// TIA Portal project "CGS1218_000_40" (V16)

(* hardware
DEVICE "SIMATIC 300"  S7-300 station
   slot 0: "Rack 0"  Rail  6ES7 390-1***0-0AA0
   slot 2: "CPU 317-2 PN/DP"  Unspecific CPU S7 300  6ES7 3XX-XXXXX-XXXX
DEVICE "SLIO_SLAVE"  S7-300 station
   slot 0: "Rack 0"  Rail  6ES7 390-1***0-0AA0
   slot 2: "CPU 315-2 PN/DP"  Unspecific CPU S7 300  6ES7 3XX-XXXXX-XXXX
DEVICE "Rack 0"  S7-300 station
   slot 0: "Rail_0"  Rail  6ES7 390-1***0-0AA0
   slot 2: "Mig_PVA_AWL"  Unspecific CPU S7 300  6ES7 3XX-XXXXX-XXXX
*)

// ===== PLC "CPU 317-2 PN/DP"  Unspecific CPU S7 300 =====
// protected blocks, not shown: "AG_LRECV_LF", "AG_LSEND_LF", "AG_RECV", "AG_SEND", "DCO_ReadDriveParameter", "DCO_WriteDriveParameter", "GLOBAL_DP_DIAG", "IO_LINK_DEVICE", "IO_LINK_MASTER"

VAR_GLOBAL   // PLC tag table "STEP7 classic symbols"
   "HDI_LS_FCH_LFT_DN" AT %I32.1 : Bool;   // HDI def M 88.1: limit switch furnace chamber lift down
   "HDI_LS_GCH_BEL_DN" AT %I274.7 : Bool;   // HDI def M 97.7: limit switch gate chamber bellow in lower position
   "HDO_XT_CLP_BLW_BRK" AT %Q275.2 : Bool;   // HDO def M 164.2: Brake crystal clamp below
   "HDO_XT_CLP_BLW_CL" AT %Q275.1 : Bool;   // HDO def M 164.1: Motor crystal clamp below close
   "HDO_XT_CLP_BLW_OP" AT %Q275.0 : Bool;   // HDO def M 164.0: Motor crystal clamp below open
   "HDO_XT_CLP_BLW_RST" AT %Q275.3 : Bool;   // HDO def M 164.3: Reset controller crystal clamp below
   "HDO_XT_CLP_TILT_BRK" AT %Q274.2 : Bool;   // HDO def M 163.2: Motor crystal clamp tilt brake
   "HDO_XT_CLP_TILT_BW" AT %Q274.0 : Bool;   // HDO def M 163.0: Motor crystal clamp tilt backwards
   "HDO_XT_CLP_TILT_FW" AT %Q274.1 : Bool;   // HDO def M 163.1: Motor crystal clamp tilt forwards (75?
   "HDO_XT_DRP_OUT_PRT_CL" AT %Q224.6 : Bool;   // HDO def M 150.6: Valve block close crystal drop out protection
   "HDO_XT_DRP_OUT_PRT_OP" AT %Q224.7 : Bool;   // HDO def M 150.7: Valve block open crystal drop out protection
   "HDO_XT_HDL_LFT_ENB" AT %Q272.7 : Bool;   // HDO def M 160.7: controller enable crystal handling lift
   "HDO_XT_HDL_SLID_BW" AT %Q273.7 : Bool;   // HDO def M 161.7: Motor crystal handling slider backwards
   "HDO_XT_HDL_SLID_FW" AT %Q273.6 : Bool;   // HDO def M 161.6: Motor crystal handling slider forwards
   "HDO_XT_HDL_SW_ENB" AT %Q273.0 : Bool;   // HDO def M 161.0: controller enable crystal handling swivel
   "HDO_XT_HDL_SW_LOCK" AT %Q225.4 : Bool;   // HDO def M 151.4: Valve block xtal handling swivel lock close (145?
   "HDO_XT_HDL_SW_UNLOCK" AT %Q225.5 : Bool;   // HDO def M 151.5: Valve block xtal handling swivel lock open (145?
   "HDO_XT_LFT_ENB" AT %Q272.6 : Bool;   // HDO def M 160.6: controller enable crystal lift
   "SM_TMR_PWR_FAIL_5S" AT %T150 : Timer;   // main line power fail 5 sec
   "STA_ITL_CAUSE" AT %MW20 : Word;
   "STA_ITL_CAUSE_DLY" AT %MW22 : Int;
   "STA_ITL_NO" AT %MB20 : Byte;
   "STA_ITL_STAT" AT %MB21 : Byte;
   "P_STA_WTR_VAC_BYP" AT %IW2194 : Word;
   "P_STA_WTR_BCH" AT %IW2164 : Word;
   "P_STA_WTR_CFT_B" AT %IW2188 : Word;
   "P_STA_WTR_CR_SFT" AT %IW2020 : Word;
   "P_STA_WTR_CUR_FEED" AT %IW2182 : Word;
   "P_STA_WTR_FCH" AT %IW2146 : Word;
   "P_STA_WTR_GCH" AT %IW2050 : Word;
   "P_STA_WTR_GCH_ADDS" AT %IW2086 : Word;
   "P_STA_WTR_GCH_H" AT %IW2068 : Word;
   "P_STA_WTR_GCH_V" AT %IW2074 : Word;
   "P_BM_MAG_ACT_CUR" AT %IW868 : Word;
   "P_BM_MAG_ACT_TMP_COIL_A1" AT %IW872 : Word;
   "P_BM_MAG_ACT_TMP_COIL_A2" AT %IW874 : Word;
   "P_BM_MAG_ACT_TMP_COIL_B1" AT %IW876 : Word;
   "P_BM_MAG_ACT_TMP_COIL_B2" AT %IW878 : Word;
   "P_BM_MAG_ACT_TMP_SHLD" AT %IW880 : Word;
   "P_BM_MAG_ACT_VLT" AT %IW870 : Word;
   "P_BM_MAG_CTRL" AT %QB864 : Byte;
   "P_BM_MAG_SET_CUR" AT %QW865 : Word;
   "P_BM_MAG_STAT" AT %IB864 : Byte;
   "P_BM_MAG_STAT2" AT %IW865 : Word;
   "P_BM_MAG_STAT3" AT %IB867 : Byte;
   "BM_MCC_OFF_TME" AT %T132 : Timer;   // melt contact control off time
   "HDI_ACC_UPS_24V_NRM" AT %I89.7 : Bool;   // HDI def M 93.7: ACC UPS Alarm
   "HDI_ACC_WTR_FLW_IN_OK" AT %I88.4 : Bool;   // HDI def M 92.4: ACC input waterflow ok
   "HDI_ACC_WTR_FLW_OUT_OK" AT %I88.3 : Bool;   // HDI def M 92.3: ACC output waterflow ok
   "HDI_ACC_WTR_TMP_OUT_OK" AT %I88.5 : Bool;   // HDI def M 92.5: ACC output watertemp. Ok
   "HDI_CB_FLT_AC230V" AT %I16.3 : Bool;   // HDI def M 72.3: fault circuit breakers AC 230V 1=OK
   "HDI_CB_FLT_AC400V_K2" AT %I16.1 : Bool;   // HDI def M 72.1: fault circuit breakers AC 400V 1=OK
   "HDI_CB_FLT_AC400V_K5" AT %I34.0 : Bool;   // HDI def M 90.0: fault circuit breakers AC 400V +K5 1=OK
   "HDI_CB_FLT_AC400V_K8" AT %I277.6 : Bool;   // HDI def M 100.6: fault circuit breakers AC 400V 1=OK
   "HDI_CB_FLT_DC24V_K2" AT %I16.0 : Bool;   // HDI def M 72.0: fault circuit breakers DC 24V 1=OK
   "HDI_CB_FLT_DC24V_K5" AT %I34.1 : Bool;   // HDI def M 90.1: fault circuit breakers DC 24V +K5 1=OK
   "HDI_CB_FLT_DC24V_K8" AT %I277.7 : Bool;   // HDI def M 100.7: fault circuit breakers DC 24V 1=OK
   "HDI_COMP_AIR_2_OK" AT %I35.7 : Bool;   // HDI def M 91.7: pressure switch compressed air 2 (ACC) ok
   "HDI_COMP_AIR_OK" AT %I35.6 : Bool;   // HDI def M 91.6: pressure switch compressed air ok
   "HDI_DPH_RPT_DET_OK" AT %I90.0 : Bool;   // HDI def M 94.0: ACC Diaphraghm rupture detector OK
   "HDI_EMO" AT %I17.3 : Bool;   // HDI def M 73.3: Emergency off (1=ok)
   "HDI_EMS" AT %I17.4 : Bool;   // HDI def M 73.4: Emergency stop handling drives (1=ok)
   "HDI_MP_ENB_K5" AT %I35.3 : Bool;   // HDI def M 91.3: Mobile panel agree button +K5
   "HDI_MP_ENB_K8" AT %I279.6 : Bool;   // HDI def M 102.6: Mobile panel agree button +K8
   "HDI_MP_ENB_K9" AT %I279.7 : Bool;   // HDI def M 102.7: Mobile panel agree button +K9
   "HDI_OIL_LVL_CR_SFT" AT %I35.0 : Bool;   // HDI def M 91.0: Crucible shaft min. oil level
   "HDI_OIL_LVL_XT_SFT" AT %I279.1 : Bool;   // HDI def M 102.1: Crystal shaft min. oil level
   "HDI_OV_PRS_1_FLT" AT %I88.6 : Bool;   // HDI def M 92.6: ACC overpressure 1 error/fault
   "HDI_OV_PRS_2_FLT" AT %I88.7 : Bool;   // HDI def M 92.7: ACC overpressure 2 error/fault
   "HDI_P1_FLT" AT %I18.1 : Bool;   // HDI def M 74.1: pump unit (P1) error
   "HDI_P1_IS_ON" AT %I18.2 : Bool;   // HDI def M 74.2: pump unit (P1) running
   "P_BM_UP_FCH_SW_ENC_REF" AT %QD1184 : DWord;   // Setpoint reference position upper furnace chamber swivel
   "BM_VAC_TMR_APS_BY_FIL" AT %T102 : Timer;   // Timer for delayed APS bypass filter
   "BM_VAC_TMR_APS_FCH" AT %T101 : Timer;   // Timer for delayed APS furnace
   "BM_VAC_TMR_APS_FDR" AT %T99 : Timer;   // Timer for delayed APS feeder
   "BM_VAC_TMR_APS_FIL" AT %T98 : Timer;   // Timer for delayed APS main filter
   "BM_VAC_TMR_APS_GCH" AT %T100 : Timer;   // Timer for delayed APS gate
   "BM_VAC_TMR_V2_ON" AT %T104 : Timer;   // Timer for delayed opening V2 after P1 on
   "BM_VAC_TMR_V3_ON" AT %T105 : Timer;   // Timer for delayed opening V3 after P3 on
   "HDI_LS_V3_OP" AT %I280.0 : Bool;   // HDI def M 103.0: valve position V3 open
   "HDI_LS_V7_CLN_POS" AT %I274.5 : Bool;   // HDI def M 97.5: limit switch gate valve V7 in cleaning position
   "HDI_LS_V7_DN" AT %I274.1 : Bool;   // HDI def M 97.1: limit switch gate valve V7 in lower position
   "HDI_LS_V7_FLP_OP" AT %I274.4 : Bool;   // HDI def M 97.4: limit switch gate valve V7 flap open
   "HDI_LS_V7_SW_IN" AT %I274.2 : Bool;   // HDI def M 97.2: limit switch gate valve V7 swiveled in
   "HDI_LS_V7_SW_OUT" AT %I274.3 : Bool;   // HDI def M 97.3: limit switch gate valve V7 swiveled out
   "HDO_SPARE_18_4" AT %Q18.4 : Bool;   // HDO def M 138.4: spare digital output
   "HDO_SPARE_18_5" AT %Q18.5 : Bool;   // HDO def M 138.5: spare digital output
   "HDO_SPARE_18_6" AT %Q18.6 : Bool;   // HDO def M 138.6: spare digital output
   "HDO_SPARE_18_7" AT %Q18.7 : Bool;   // HDO def M 138.7: spare digital output
   "HDO_SPARE_226_2" AT %Q226.2 : Bool;   // HDO def M 152.2: Valve block spare output
   "HDO_SPARE_226_3" AT %Q226.3 : Bool;   // HDO def M 152.3: Valve block spare output
   "HDO_SPARE_226_4" AT %Q226.4 : Bool;   // HDO def M 152.4: Valve block spare output
   "HDO_SPARE_226_5" AT %Q226.5 : Bool;   // HDO def M 152.5: Valve block spare output
   "HDO_SPARE_226_6" AT %Q226.6 : Bool;   // HDO def M 152.6: Valve block spare output
   "HDO_SPARE_226_7" AT %Q226.7 : Bool;   // HDO def M 152.7: Valve block spare output
   "P_BM_ACT_WTR_TMP_PWR_CAB" AT %IW2024 : Word;   // HAI def MW 356: actual water temperature high current cables Main K18
   "P_BM_ACT_WTR_TMP_PWR_CAB2" AT %IW2030 : Word;   // HAI def MW 347: actual water temperature current feed throughs B K19
   "P_BM_ACT_WTR_TMP_SOC_BCH" AT %IW2174 : Word;   // HAI def MW 329: actual water temperature socket bottom chamber K13
   "P_BM_ACT_WTR_TMP_TCH" AT %IW2090 : Word;   // HAI def MW 239: actual water temperature top chamber K07
   "P_BM_ACT_WTR_TMP_TEC_FLG" AT %IW2114 : Word;   // HAI def MW 275: actual water temperature technolity chamber K08
   "P_BM_ACT_WTR_TMP_UP_FCH" AT %IW2132 : Word;   // HAI def MW 338: actual water temperature upper furnace chamber K10
   "P_BM_ACT_WTR_TMP_VPTS" AT %IW2078 : Word;   // HAI def MW 291: actual water temperature view ports K06
   "P_BM_ACT_WTR_TMP_XT_SFT" AT %IW2036 : Word;   // HAI def MW 246: actual water temperature seed shaft K02
   "DP_DEATV_ERR_CODE_N9" AT %MW62 : Int;   // DP Slave +N9 (active cooling) deactivation error code
   "DP_DEATV_TSK_RUN_N9" AT %M52.5 : Bool;   // DP Slave +N9 (active cooling) deactivation busy flag
   "HDO_MAG_LFT_UP" AT %Q33.2 : Bool;   // HDO def M 143.2: Magnet lift drive upwards
   "HDO_MCC_ENB_XT" AT %Q275.5 : Bool;   // HDO def M 164.5: seed contact detection enable output (xt isolated)
   "HDO_MCC_TEST_XT" AT %Q275.4 : Bool;   // HDO def M 164.4: seed contact detection test output ( xt isolated)
   "HDO_MON_TMP_P2_RES" AT %Q17.7 : Bool;   // HDO def M 137.7: temperature monitoring pump 2 reset
   "HDO_P1_ON" AT %Q17.0 : Bool;   // HDO def M 137.0: Vacuum pump 1 on (furnace chamber)
   "HDO_P1_SEAL_GAS" AT %Q17.3 : Bool;   // HDO def M 137.3: Vacuum pump 1 seal gas on
   "HDO_P2_FU_ON" AT %Q144.0 : Bool;   // HDO def M 152.0: Frequency converter P2 start
   "HDO_P2_FU_RES" AT %Q144.1 : Bool;   // HDO def M 152.1: Frequency converter P2 fault reset
   "HDI_SPARE_16_5" AT %I16.5 : Bool;   // HDI def M 72.5: spare digital input
   "HDI_SPARE_16_6" AT %I16.6 : Bool;   // HDI def M 72.6: spare digital input
   "HDI_SPARE_16_7" AT %I16.7 : Bool;   // HDI def M 72.7: spare digital input
   "HDI_SPARE_17_0" AT %I17.0 : Bool;   // HDI def M 73.0: spare digital input
   "HDI_SPARE_17_5" AT %I17.5 : Bool;   // HDI def M 73.5: spare digital input
   "HDI_SPARE_17_6" AT %I17.6 : Bool;   // HDI def M 73.6: spare digital input
   "HDI_SPARE_17_7" AT %I17.7 : Bool;   // HDI def M 73.7: spare digital input
   "HDI_SPARE_18_7" AT %I18.7 : Bool;   // HDI def M 74.7: spare digital input
   "HDI_SPARE_275_7" AT %I275.7 : Bool;   // HDI def M 98.7: spare digital input
   "HDI_SPARE_280_5" AT %I280.5 : Bool;   // HDI def M 103.5: spare digital input
   "HDI_SPARE_280_6" AT %I280.6 : Bool;   // HDI def M 103.6: spare digital input
   "HDI_SPARE_280_7" AT %I280.7 : Bool;   // HDI def M 103.7: spare digital input
   "HDI_SPARE_33_4" AT %I33.4 : Bool;   // HDI def M 89.4: spare
   "HDI_SPARE_33_5" AT %I33.5 : Bool;   // HDI def M 89.5: spare
   "HDI_SPARE_48_2" AT %I88.2 : Bool;   // HDI def M 92.2: ACC spare
   "HDI_SPARE_90_2" AT %I90.2 : Bool;   // HDI def M 94.2: ACC spare
   "P_reserve_2_X08_WTR_TMP" AT %IW2108 : Word;
   "P_reserve_3_X08_WTR_FLW" AT %IW2154 : Word;
   "HDI_LS_V2_11_OP" AT %I36.6 : Bool;   // HDI def M 105.6: limit switch valve v2.11 opened
   "HDI_LS_V2_1_CL" AT %I33.7 : Bool;   // HDI def M 89.7: valve position v2.1 fce chamber
   "HDI_LS_V2_1_OP" AT %I33.6 : Bool;   // HDI def M 89.6: valve position v2.1 fce chamber
   "HDI_LS_V3_3_CL" AT %I36.5 : Bool;   // HDI def M 105.5: limit switch valve v3.3 closed
   "HDI_LS_V3_3_OP" AT %I36.4 : Bool;   // HDI def M 105.4: limit switch valve v3.3 opened
   "HDI_LS_V3_4_CL" AT %I36.3 : Bool;   // HDI def M 105.3: limit switch valve v3.4 closed
   "HDI_LS_V3_4_OP" AT %I36.2 : Bool;   // HDI def M 105.2: limit switch valve v3.4 opened
   "HDI_LS_V3_CL" AT %I280.1 : Bool;   // HDI def M 103.1: Valve position V3 closed
   "MELT_CON_DETECT_DLY" AT %T134 : Timer;   // melt contact control delay timer
   "SysEdgeFlag400ms" AT %M3.4 : Bool;   // System Cycle: Edge Flag 400 ms
   "SysEdgeFlag500ms" AT %M3.6 : Bool;   // System Cycle: Edge Flag 500 ms
   "SysEdgeFlag800ms" AT %M4.0 : Bool;   // System Cycle: Edge Flag 800 ms
   "SysImpFlag100ms" AT %M3.1 : Bool;   // System Cycle: Impuls Flag 100 ms
   "SysImpFlag1_6s" AT %M4.5 : Bool;   // System Cycle: Impuls Flag 1600 ms
   "SysImpFlag1s" AT %M4.3 : Bool;   // System Cycle: Impuls Flag 1000 ms
   "SysImpFlag200ms" AT %M3.3 : Bool;   // System Cycle: Impuls Flag 200 ms
   "SysImpFlag2s" AT %M4.7 : Bool;   // System Cycle: Impuls Flag 2000 ms
   "SysImpFlag400ms" AT %M3.5 : Bool;   // System Cycle: Impuls Flag 400 ms
   "SysImpFlag500ms" AT %M3.7 : Bool;   // System Cycle: Impuls Flag 500 ms
   "SysImpFlag800ms" AT %M4.1 : Bool;   // System Cycle: Impuls Flag 800 ms
   "SysLog0" AT %M0.0 : Bool;   // System: Logical 0
   "SysLog1" AT %M0.1 : Bool;   // System: Logical 1
   "SysTick100ms" AT %M1.0 : Bool;   // System Tick: 100 ms
   "P_BM_PWR_SPL_2_SET_PWR" AT %QD902 : Real;   // setpoint power heater 2
   "P_BM_PWR_SPL_CTRL" AT %QB896 : Byte;   // Heater on
   "P_BM_PWR_SPL_CTRL_W" AT %QW896 : Word;   // power supply control word
   "P_BM_PWR_SPL_STAT" AT %IW896 : Word;   // statusword 1 power supply
   "P_BM_PWR_SPL_STAT2" AT %IW898 : Word;   // statusword 2 power supply
   "P_BM_PWR_SPL_STAT3" AT %IW900 : Word;   // statusword 3 power supply
   "P_BM_PWR_SPL_STAT4" AT %IW902 : Word;   // statusword 4 power supply
   "P_BM_PWR_SPL_STAT5" AT %IW904 : Word;   // statusword 5 power supply
   "P_BM_PWR_SPL_STAT6" AT %IW906 : Word;   // statusword 6 power supply
   "P_BM_PWR_SPL_STAT7" AT %IW908 : Word;   // statusword 7 power supply
   "HDI_LS_MAG_LFT_UP" AT %I34.2 : Bool;   // HDI def M 90.2: limit switch magnet lift up
   "HDI_LS_TCH_DN" AT %I273.0 : Bool;   // HDI def M 96.0: limit switch top chamber in lower position
   "HDI_LS_TCH_SW_CLN" AT %I273.2 : Bool;   // HDI def M 96.2: limit switch top chamber swivelled in cleaning pos
   "HDI_LS_TCH_SW_IN" AT %I273.1 : Bool;   // HDI def M 96.1: limit switch top chamber swivelled in
   "HDI_LS_TCH_SW_LOCK" AT %I273.4 : Bool;   // HDI def M 96.4: limit switch top chamber swivel locked
   "HDI_LS_TCH_SW_OUT" AT %I273.3 : Bool;   // HDI def M 96.3: limit switch top chamber swivelled out
   "HDI_LS_TCH_TILT_0" AT %I273.5 : Bool;   // HDI def M 96.5: limit switch top chamber tilt 0?horizental
   "HDI_LS_TCH_TILT_30" AT %I273.6 : Bool;   // HDI def M 96.6: limit switch top chamber tilt 30?Cleaning position
   "HDI_LS_TCH_UP" AT %I272.7 : Bool;   // HDI def M 95.7: limit switch top chamber in upper position
   "HDI_LS_TEC_FLG_DN" AT %I32.4 : Bool;   // HDI def M 88.4: limit switch technolgy flange down
   "HDO_HOR_OPP_K2" AT %Q16.0 : Bool;   // HDO def M 136.0: Horn +K2
   "HDO_HOR_OPP_K8" AT %Q272.0 : Bool;   // HDO def M 160.0: Horn +K8
   "HDO_HOR_OPP_K9" AT %Q276.3 : Bool;   // HDO def M 165.3: Horn +K9
   "HDO_HTR_PWR_ON" AT %Q17.5 : Bool;   // HDO def M 137.4: Heater power supply on
   "P_BM_ACT_GAS_FLW_MFC_1" AT %ID1376 : Real;   // actual gas flow from mfc with profinet interface
   "P_BM_ACT_GAS_FLW_MFC_2" AT %ID1408 : Real;   // actual gas flow from mfc with profinet interface
   "P_BM_ACT_WTR_FLW_VAC_BYP" AT %IW2190 : Word;   // actual water flow vacuum bypass tube
   "P_BM_ACT_WTR_FLW_BCH" AT %IW2160 : Word;   // HAI def MW 309: actual water flow bottom chamber K12
   "P_BM_ACT_WTR_FLW_CFT_B" AT %IW2184 : Word;   // HAI def MW 235: actual water flow current feed throught Bot K15
   "P_BM_ACT_WTR_FLW_CFT_M" AT %IW2178 : Word;   // HAI def MW 217: actual water flow current feed throught Main K14
   "P_BM_ACT_WTR_FLW_CR_SFT" AT %IW2016 : Word;   // HAI def MW 208: actual water flow crucible shaft K17
   "P_BM_ACT_WTR_FLW_FCH" AT %IW2142 : Word;   // HAI def MW 300: actual water flow furnace chamber K11
   "P_BM_ACT_WTR_FLW_GCH" AT %IW2046 : Word;   // HAI def MW 262: actual water flow gate chamber K03
   "P_BM_ACT_WTR_FLW_GCH_ADDS" AT %IW2082 : Word;   // HAI def MW 298: actual water flow chamber parts, view ports K24
   "HDI_XT_ROT_CAM_TRG" AT %I279.5 : Bool;   // HDI def M 102.5: limit switch xtal rotation camera trigger
   "HDO_ACC_ALM_LT_1" AT %Q88.4 : Bool;   // HDO def M 146.4: ACC Blitzlicht Kasten
   "HDO_ACC_ALM_LT_2" AT %Q88.6 : Bool;   // HDO def M 146.6: ACC Blitzlicht Bedienpult
   "HDO_ACC_ALM_SND_1" AT %Q88.5 : Bool;   // HDO def M 146.5: ACC Sirene Kasten
   "HDO_ACC_ALM_SND_2" AT %Q88.7 : Bool;   // HDO def M 146.7: ACC Sirene Bedienpult
   "HDO_ACC_SC_HTR_RST" AT %Q88.1 : Bool;   // HDO def M 146.1: ACC Heizung RESET
   "HDO_ACC_SC_HTR_STR" AT %Q88.0 : Bool;   // HDO def M 146.0: ACC Heizung START
   "HDO_ACC_SC_WTR_RST" AT %Q88.3 : Bool;   // HDO def M 146.3: ACC K黨lwasser RESET
   "HDO_ACC_SC_WTR_STR" AT %Q88.2 : Bool;   // HDO def M 146.2: ACC K黨lwasser START
   "HDO_BEL_LFT_ENB" AT %Q276.2 : Bool;   // HDO def M 165.2: controller enable gate bellow lift
   "HDO_BRK_MAG_LFT" AT %Q33.4 : Bool;   // HDO def M 143.4: Brake magnet lift
   "HDO_CR_LFT_ENB" AT %Q32.6 : Bool;   // HDO def M 142.6: controller enable crucible lift
   "HDO_CR_ROT_ENB" AT %Q32.5 : Bool;   // HDO def M 142.5: controller enable crucible rotation
   "HDO_FCH_HOOK_HOME" AT %Q96.0 : Bool;   // HDO def M 150.0: Valve block lower furnace chamber hook unlocking
   "HDO_V24" AT %Q224.5 : Bool;   // HDO def M 150.5: Valve block V24 valve argon gas inlet feeder
   "HDO_V25" AT %Q96.5 : Bool;   // HDO def M 150.5: Valve block argon inlet pressure storage tank, V25 open
   "HDO_V2_1" AT %Q96.6 : Bool;   // HDO def M 150.6: Valve block vacuum valve, V2.1 open
   "HDO_V2_11" AT %Q97.7 : Bool;   // HDO def M 151.7: Valve block vacuum valve, V2.11 open
   "HDO_V3" AT %Q224.3 : Bool;   // HDO def M 150.3: Valve block V3 vacuum valve (gate chamber)
   "HDO_V3_2" AT %Q224.4 : Bool;   // HDO def M 150.4: Valve block V3.2 vacuum valve feeder
   "HDO_V3_3" AT %Q97.6 : Bool;   // HDO def M 151.6: Valve block vacuum valve, V3.3 open
   "HDO_V3_4" AT %Q97.5 : Bool;   // HDO def M 151.5: Valve block vacuum valve, V3.4 open
   "HDO_V4" AT %Q224.0 : Bool;   // HDO def M 150.0: Valve block V4 valve argon gas inlet (gate chamber)
   "HDO_V5" AT %Q224.1 : Bool;   // HDO def M 150.1: Valve block V5 valve argon gas inlet controlled (gch)
   "HDO_V6" AT %Q224.2 : Bool;   // HDO def M 150.2: Valve block V6 valve argon gas inlet controlled (Fch)
   "HDO_V9_2" AT %Q97.3 : Bool;   // HDO def M 151.3: Valve block ventiliation valve vaccum line gate, V9_2
   "HDO_XT_CLP_ABV_BRK" AT %Q274.5 : Bool;   // HDO def M 163.5: Brake crystal clamp above
   "HDO_XT_CLP_ABV_CL" AT %Q274.4 : Bool;   // HDO def M 163.4: Motor crystal clamp above close
   "HDO_XT_CLP_ABV_OP" AT %Q274.3 : Bool;   // HDO def M 163.3: Motor crystal clamp above open
   "HDO_XT_CLP_ABV_RST" AT %Q274.6 : Bool;   // HDO def M 163.6: Reset controller crystal clamp above
   "SM_TMR_PWR_FAIL_3M" AT %T151 : Timer;   // main line power fail 3 min
   "P_BM_FDR_STAT" AT %ID1504 : DWord;
   "P_BM_FDR_VIB_FRQ" AT %QD1508 : Real;
   "P_BM_HTR_1_ETH_CTRL" AT %QB1044 : Byte;   // heater 1 earthing monitoring control byte
   "P_BM_HTR_1_ETH_STA" AT %IB1060 : Byte;   // heater 1 earthing monitoring status byte
   "P_BM_HTR_2_ETH_CTRL" AT %QB1049 : Byte;   // heater 2 earthing monitoring control byte
   "P_BM_HTR_2_ETH_STA" AT %IB1065 : Byte;   // heater 2 earthing monitoring status byte
   "P_BM_LO_FCH_SW_ENC_POS" AT %ID1216 : DWord;   // actual encoder position lower furnace chamber swivel
   "P_BM_LO_FCH_SW_ENC_REF" AT %QD1216 : DWord;   // Setpoint reference position lower furnace chamber swivel
   "P_HAI_TRV_PRS_FIL_1" AT %IW588 : Word;   // HAI def MW 204: actual pressure value main filter
   "P_HAI_TRV_PRS_FIL_2" AT %IW590 : Word;   // HAI def MW 206: actual pressure value bypass filter
   "HAO_SPARE" AT %MW304 : Word;   // HAO def MW 304: spare
   "P_HAO_TRV_SET_POS" AT %QW576 : Word;   // HAO def MW 300: setpoint throttle valve 1 position
   "P_HAO_TRV_SET_POS_1" AT %QW578 : Word;   // HAO def MW 302: setpoint throttle valve 1.1 position
   "HDI_ACC_CB_FLT_AC230V" AT %I90.1 : Bool;   // HDI def M 94.1: Fault circuit breakers AC 230V
   "HDI_ACC_CB_FLT_DC24V" AT %I89.5 : Bool;   // HDI def M 93.5: ACC 24V circuit breaker ok
   "HDI_ACC_FCH_OV_PRS_1" AT %I88.0 : Bool;   // HDI def M 92.0: ACC furnace overpressure 1
   "HDI_ACC_FCH_OV_PRS_2" AT %I88.1 : Bool;   // HDI def M 92.1: ACC furnace overpressure 2
   "HDI_ACC_KEY_RST" AT %I89.4 : Bool;   // HDI def M 93.4: ACC reset key
   "HDI_ACC_SC_HTR_ATV" AT %I89.3 : Bool;   // HDI def M 93.3: ACC safety circuit
   "HDI_ACC_SC_HTR_OK" AT %I89.2 : Bool;   // HDI def M 93.2: ACC safety circuit
   "HDI_ACC_SC_WTR_ATV" AT %I89.1 : Bool;   // HDI def M 93.1: ACC safety circuit
   "HDI_ACC_SC_WTR_OK" AT %I89.0 : Bool;   // HDI def M 93.0: ACC safety circuit
   "HDI_ACC_UPS_24V_ALM" AT %I89.6 : Bool;   // HDI def M 93.6: ACC UPS OK Normal
   "HDO_TCH_SW_LOCK" AT %Q225.0 : Bool;   // HDO def M 151.0: Valve block top chamber swivel lock close
   "HDO_TCH_SW_UNLOCK" AT %Q225.1 : Bool;   // HDO def M 151.1: Valve block top chamber swivel lock open
   "VIMP_LS_XT_HDL_SW_LOCK" AT %MW36 : Int;
   "P_reserve_1_X07_WTR_FLW" AT %IW2052 : Word;
   "P_reserve_1_X07_WTR_TMP" AT %IW2054 : Word;
   "P_reserve_1_X08_WTR_FLW" AT %IW2058 : Word;
   "P_reserve_1_X08_WTR_TMP" AT %IW2060 : Word;
   "P_reserve_2_X06_WTR_FLW" AT %IW2094 : Word;
   "P_reserve_2_X06_WTR_TMP" AT %IW2096 : Word;
   "P_reserve_2_X07_WTR_FLW" AT %IW2100 : Word;
   "P_reserve_2_X07_WTR_TMP" AT %IW2102 : Word;
   "P_reserve_2_X08_WTR_FLW" AT %IW2106 : Word;
   "P_BM_XT_HDL_LFT_FU_POS" AT %ID1696 : Real;   // actual frequenz converter position Crystal handling lift
   "P_BM_XT_HDL_SW_ENC_POS" AT %ID1248 : DWord;   // actual encoder position Crystal handling swivel
   "P_BM_XT_HDL_SW_ENC_REF" AT %QD1248 : DWord;   // Setpoint reference position Crystal handling swivel
   "HDI_LS_XT_TOP_POS" AT %I279.3 : Bool;   // HDI def M 102.3: limit switch crystal shaft in top position
   "HDI_MAG_LFT_SDL_NUT1" AT %I34.5 : Bool;   // HDI def M 90.5: safety limit switch magnet lift spindle nut 1
   "HDI_MAG_LFT_SDL_NUT2" AT %I34.6 : Bool;   // HDI def M 90.6: safety limit switch magnet lift spindle nut 2
   "HDI_MAG_LFT_SDL_NUT3" AT %I34.7 : Bool;   // HDI def M 90.7: safety limit switch magnet lift spindle nut 3
   "HDI_MCC_CONTACT_XT" AT %I279.0 : Bool;   // HDI def M 102.0: seed contact detection (xt isolated)
   "HDI_MON_TMP_P1" AT %I18.6 : Bool;   // HDI def M 74.6: temperature monitoring P1
   "HDI_MON_TMP_P2" AT %I18.5 : Bool;   // HDI def M 74.5: temperature monitoring P2
   "HDO_FCH_HOOK_WORK" AT %Q96.1 : Bool;   // HDO def M 150.1: Valve block lower furnace chamber hook locking
   "HDO_FCH_LFT_ENB" AT %Q33.1 : Bool;   // HDO def M 143.1: controller enable lower chamber parts lift
   "HDI_SPARE_90_3" AT %I90.3 : Bool;   // HDI def M 94.3: ACC spare
   "HDI_SPARE_90_4" AT %I90.4 : Bool;   // HDI def M 94.4: ACC spare
   "HDI_SPARE_90_5" AT %I90.5 : Bool;   // HDI def M 94.5: ACC spare
   "HDI_SPARE_90_6" AT %I90.6 : Bool;   // HDI def M 94.6: ACC spare
   "HDI_SPARE_90_7" AT %I90.7 : Bool;   // HDI def M 94.7: ACC spare
   "HDI_TEC_FLG_SDL_NUT" AT %I32.5 : Bool;   // HDI def M 88.5: safety limit switch technolgy flange lift spindle nut
   "HDI_UPS_24V_ALM" AT %I17.1 : Bool;   // HDI def M 73.1: alarm dc-usv
   "HDI_UPS_24V_NRM" AT %I17.2 : Bool;   // HDI def M 73.2: main line ready buffered dc-usv
   "HDI_XT_DRP_OUT_PRT_1_CL" AT %I277.2 : Bool;   // HDI def M 100.2: crystal drop out protection 1 closed (upper left side)
   "HDI_XT_DRP_OUT_PRT_1_OP" AT %I277.3 : Bool;   // HDI def M 100.3: crystal drop out protection 1 opened (upper left side)
   "HDI_XT_DRP_OUT_PRT_2_CL" AT %I277.4 : Bool;   // HDI def M 100.4: crystal drop out protection 2 closed (upper right side)
   "HDI_XT_DRP_OUT_PRT_2_OP" AT %I277.5 : Bool;   // HDI def M 100.5: crystal drop out protection 2 opened (upper right side)
   "HDI_XT_DRP_OUT_PRT_3_CL" AT %I278.0 : Bool;   // HDI def M 101.0: crystal drop out protection 3 closed (lower left side)
   "HDI_XT_DRP_OUT_PRT_3_OP" AT %I278.1 : Bool;   // HDI def M 101.1: crystal drop out protection 3 opened (lower left side)
   "HDI_XT_DRP_OUT_PRT_4_CL" AT %I278.2 : Bool;   // HDI def M 101.2: crystal drop out protection 4 closed (lower right side)
   "HDI_XT_DRP_OUT_PRT_4_OP" AT %I278.3 : Bool;   // HDI def M 101.3: crystal drop out protection 4 opened (lower right side)
   "HDO_TCH_TILT_ENB" AT %Q275.7 : Bool;   // HDO def M 164.7: controller enable top chamber tilt
   "HDO_TEC_FLG_LFT_ENB" AT %Q33.0 : Bool;   // HDO def M 143.0: controller enable techn chamber lift
   "HDO_TEC_FLG_SW_BRK" AT %Q96.4 : Bool;   // HDO def M 150.4: Valve block tech. flange swivel release brake
   "HDO_UP_FCH_SW_BRK" AT %Q96.2 : Bool;   // HDO def M 150.2: Valve block upper chamber swivel release brake
   "HDO_V10" AT %Q17.6 : Bool;   // HDO def M 137.6: Vacuum pump 1 secuvac valve V10 on
   "HDO_V19" AT %Q97.0 : Bool;   // HDO def M 151.0: Valve block extraktion valve filter, V19 open
   "HDO_V1_1_CL" AT %Q34.1 : Bool;   // HDO def M 144.1: V1.1 close
   "HDO_V1_1_OP" AT %Q34.0 : Bool;   // HDO def M 144.0: V1.1 open
   "HDO_V1_CL" AT %Q32.1 : Bool;   // HDO def M 142.1: V1 close
   "HDO_V1_OP" AT %Q32.0 : Bool;   // HDO def M 142.0: V1 open
   "HDO_V20" AT %Q97.1 : Bool;   // HDO def M 151.1: Valve block air valve filter, V20 open
   "HDO_V21" AT %Q96.7 : Bool;   // HDO def M 150.7: Valve block air valve vacuum pipe, V21+V21.1 open
   "HDO_V22" AT %Q97.2 : Bool;   // HDO def M 151.2: Valve block argon valve filter, V22 open
   "HDO_V22_1" AT %Q97.4 : Bool;   // HDO def M 151.4: Valve block argon valve bypass filter, V22.1 open
   "P_BM_ETH_FLT_MON_UIST2" AT %IW1061 : Int;   // Bottom heater earth fault monitoring voltage in
   "P_BM_FCH_ENC_POS" AT %ID1152 : DWord;   // actual encoder position furnace chamber lift
   "P_BM_FCH_ENC_REF" AT %QD1152 : DWord;   // Setpoint reference position furnace chamber lift
   "P_BM_FDR_ACT_CRG_LVL" AT %ID1520 : Real;
   "P_BM_FDR_ACT_TUBE_POS" AT %ID1516 : Real;
   "P_BM_FDR_ACT_VIB" AT %ID1512 : Real;
   "P_BM_FDR_CTRL" AT %QD1504 : DWord;
   "P_BM_FDR_PCR_ACT_PRS" AT %ID1508 : Real;
   "P_HAI_ACC_WTR_SPL_PRS" AT %IW808 : Word;   // HAI def MW 266: ACC water supply inlet pressure
   "P_HAI_ACC_WTR_TMP" AT %IW800 : Word;   // HAI def MW 258: ACC water temp.
   "P_HAI_FCH_BAR_ACT_PRS_100" AT %IW1548 : Word;   // HAI def MW 198: actual vacuum gauge furnace chamber 100 mbar
   "P_HAI_FCH_PCR_ACT_PRS" AT %IW1546 : Word;   // HAI def MW 200: actual vacuum gauge furnace chamber 5xe-4...1500 mbar
   "P_HAI_GCH_PCR_ACT_PRS" AT %IW1544 : Word;   // HAI def MW 242: actual vacuum gauge gate chamber 5xe-4...1500 mbar
   "P_HAI_PYR_ACT_HTR_1_TMP" AT %IW480 : Word;   // HAI def MW 250: actual temperature main heater
   "P_HAI_PYR_ACT_MELT_TMP" AT %IW1536 : Word;   // HAI def MW 280: actual temperature melt
   "HAI_SPARE" AT %MW270 : Word;   // HAI def MW 270: spare
   "P_HAI_SPARE_1538" AT %IW1538 : Word;   // HAI def MW 282: spare analog output (4..20 mA)
   "P_HAI_SPARE_1540" AT %IW1540 : Word;   // HAI def MW 284: spare analog output (4..20 mA)
   "P_HAI_SPARE_1542" AT %IW1542 : Word;   // HAI def MW 286: spare analog output (4..20 mA)
   "P_HAI_ACT_PRS_AR_VSL" AT %IW482 : Word;   // HAI def MW 252: actual pressure argon storage tank
   "P_HAI_SPARE_484" AT %IW484 : Word;   // HAI def MW 254: spare analog output (4..20 mA)
   "P_HAI_SPARE_486" AT %IW486 : Word;   // HAI def MW 256: spare analog output (4..20 mA)
   "P_HAI_TRV_ACT_POS" AT %IW576 : Word;   // HAI def MW 192: actual throttle valve position
   "P_HAI_TRV_ACT_POS_1" AT %IW578 : Word;   // HAI def MW 194: actual throttle valve 1.1 position
   "HDO_SPARE_273_3" AT %Q273.3 : Bool;   // HDO def M 161.3: spare digital output
   "HDO_SPARE_273_4" AT %Q273.4 : Bool;   // HDO def M 161.4: spare digital output
   "HDO_SPARE_273_5" AT %Q273.5 : Bool;   // HDO def M 161.5: spare digital output
   "HDO_SPARE_32_2" AT %Q32.2 : Bool;   // HDO def M 142.2: spare digital output
   "HDI_LS_V7_UP" AT %I274.0 : Bool;   // HDI def M 97.0: limit switch gate valve V7 in upper position
   "HDI_LS_XT_CLP_CON" AT %I275.3 : Bool;   // HDI def M 98.3: limit switch crystal handling clamps connected
   "HDI_LS_XT_HDL_SW_UNLOCK" AT %I278.4 : Bool;   // HDI def M 101.4: limit switch crystal handling swivel unlocked
   "HDI_LS_XT_SFT_SRV_POS" AT %I279.2 : Bool;   // HDI def M 102.2: limit switch crystal shaft service position
   "HDI_LS_XT_SLID_BW" AT %I275.0 : Bool;   // HDI def M 98.0: limit switch crystal handling slider in home position
   "HDI_LS_XT_SLID_FW" AT %I275.1 : Bool;   // HDI def M 98.1: limit switch crystal handling slider in work position
   "HDI_LS_XT_SLID_MID" AT %I275.2 : Bool;   // HDI def M 98.2: limit switch crystal handling slider in middle position
   "NFM_LS_FCH_LFT_DN" AT %M38.2 : Bool;
   "NFM_TEC_FLG_DN" AT %M38.1 : Bool;
   "SysTick1_6s" AT %M1.6 : Bool;   // System Tick: 1600 ms
   "SysTick1s" AT %M1.5 : Bool;   // System Tick: 1000 ms
   "SysTick200ms" AT %M1.1 : Bool;   // System Tick: 200 ms
   "SysTick2s" AT %M1.7 : Bool;   // System Tick: 2000 ms
   "SysTick400ms" AT %M1.2 : Bool;   // System Tick: 400 ms
   "SysTick500ms" AT %M1.3 : Bool;   // System Tick: 500 ms
   "SysTick800ms" AT %M1.4 : Bool;   // System Tick: 800 ms
   "TI_PRESET_FCH_LFT" AT %MW26 : Int;
   "TI_PRESET_LO_FCH_SW" AT %MW30 : Int;
   "TI_PRESET_TEC_FLG" AT %MW28 : Int;
   "TI_PRESET_TEC_FLG_SW" AT %MW34 : Int;
   "TI_PRESET_UP_FCH_SW" AT %MW32 : Int;
   "TI_PRESET_XT_HDL_SW" AT %MW24 : Int;
   "P_BM_SET_GAS_FLW_MFC_1" AT %QD1376 : Real;   // gas flow setpoint for mfc with profinet interface
   "P_BM_SET_GAS_FLW_MFC_2" AT %QD1408 : Real;   // gas flow setpoint for mfc with profinet interface
   "P_BM_TEC_FLG_ENC_POS" AT %ID1088 : DWord;   // actual encoder position technology flange lift
   "P_BM_TEC_FLG_ENC_REF" AT %QD1088 : DWord;   // Setpoint reference position technology flange chamber lift
   "P_BM_TEC_FLG_SW_ENC_POS" AT %ID1120 : DWord;   // actual encoder position technolegy flange chamber swivel
   "P_BM_TEC_FLG_SW_ENC_REF" AT %QD1120 : DWord;   // Setpoint reference position technolegy flange chamber swivel
   "BM_TMR_LO_FCH_SW" AT %T52 : Timer;   // lower furnace chamber swivel opening time brake
   "BM_TMR_MAG_DRV" AT %T91 : Timer;   // delay magnet drive start
   "BM_TMR_TEC_FLG_SW" AT %T50 : Timer;   // Techn.flange swivel opening time brake
   "BM_TMR_UP_FCH_SW" AT %T51 : Timer;   // Upper furnace chamber swivel opening time brake
   "P_BM_UP_FCH_SW_ENC_POS" AT %ID1184 : DWord;   // actual encoder position upper furnace chamber swivel
   "HDI_LS_V11_COV_CL" AT %I32.7 : Bool;   // HDI def M 88.7: Cover V11 closed (isolation valve feeder)
   "HDI_LS_V11_COV_OP" AT %I32.6 : Bool;   // HDI def M 88.6: Cover V11 opened (isolation valve feeder)
   "HDI_LS_V11_OP" AT %M89.3 : Bool;   // HDI def M 89.3: V 11 open (isolation valve feeder)
   "HDI_LS_V1_1_CL" AT %I36.0 : Bool;   // HDI def M 105.0: limit switch valve v1.1 closed
   "HDI_LS_V1_1_OP" AT %I36.1 : Bool;   // HDI def M 105.1: limit switch valve v1.1 opened
   "HDI_LS_V1_CL" AT %I35.2 : Bool;   // HDI def M 91.2: V1 closed
   "HDI_LS_V1_OP" AT %I35.1 : Bool;   // HDI def M 91.1: V1 opened
   "HDI_LS_V2_11_CL" AT %I36.7 : Bool;   // HDI def M 105.7: limit switch valve v2.11 closed
   "HDO_P2_ON" AT %Q17.2 : Bool;   // HDO def M 137.2: Vacuum pump 2 on (roots furnace chamber)
   "HDO_P3_ON" AT %Q17.1 : Bool;   // HDO def M 137.1: Vacuum pump 3 on (gate chamber)
   "HDO_P3_SEAL_GAS" AT %Q17.4 : Bool;   // HDO def M 137.4: Vacuum pump 3 seal gas on
   "HDO_SPARE_144_2" AT %Q144.2 : Bool;   // HDO def M 152.2: spare digital output
   "HDO_SPARE_144_3" AT %Q144.3 : Bool;   // HDO def M 152.3: spare digital output
   "HDO_SPARE_144_4" AT %Q144.4 : Bool;   // HDO def M 152.4: spare digital output
   "HDO_SPARE_144_5" AT %Q144.5 : Bool;   // HDO def M 152.5: spare digital output
   "HDO_SPARE_144_6" AT %Q144.6 : Bool;   // HDO def M 152.6: spare digital output
   "P_BM_ACT_WTR_TMP_VAC_BYP" AT %IW2192 : Word;   // actual water temperature vacuum bypass tube
   "P_BM_ACT_WTR_TMP_BCH" AT %IW2162 : Word;   // HAI def MW 311: actual water temperature bottom chamber K12
   "P_BM_ACT_WTR_TMP_CFT_B" AT %IW2186 : Word;   // HAI def MW 237: actual water temperature current feed throught Bot K15
   "P_BM_ACT_WTR_TMP_CFT_M" AT %IW2180 : Word;   // HAI def MW 219: actual water temperature current feed throught M K14
   "P_BM_ACT_WTR_TMP_CR_SFT" AT %IW2018 : Word;   // HAI def MW 210: actual water temperature crucible shaft K17
   "P_BM_ACT_WTR_TMP_FCH" AT %IW2144 : Word;   // HAI def MW 302: actual water temperature furnace chamber K11
   "P_BM_ACT_WTR_TMP_GCH" AT %IW2048 : Word;   // HAI def MW 264: actual water temperature gate chamber K03
   "P_BM_ACT_WTR_TMP_GCH_ADDS" AT %IW2084 : Word;   // HAI def MW 230: actual water temperature chamber parts, view ports K24
   "P_BM_ACT_WTR_TMP_GCH_H" AT %IW2066 : Word;   // HAI def MW 273: actual water temperature gate chamber valve housing K04
   "P_BM_ACT_WTR_TMP_GCH_V" AT %IW2072 : Word;   // HAI def MW 282: actual water temperature gate chamber valve K05
   "P_BM_ACT_WTR_TMP_HTR" AT %IW2042 : Word;   // HAI def MW 255: actual water temperature heater power supply K20
   "P_BM_ACT_WTR_TMP_MAG_CAB" AT %IW2168 : Word;   // HAI def MW 320: actual water temperature magnet power supply K30
   "P_BM_ACT_WTR_TMP_MAG_CO1" AT %IW2150 : Word;   // HAI def MW 284: actual water temperature magnet compressor unit 1 K29
   "P_BM_ACT_WTR_TMP_MAG_CO2" AT %IW2138 : Word;   // HAI def MW 293: actual water temperature magnet compressor unit 2 K28
   "P_BM_ACT_WTR_TMP_MAG_CO3" AT %IW2126 : Word;   // HAI def MW 257: actual water temperature magnet compressor unit 3 K27
   "P_BM_ACT_WTR_TMP_MAG_CO4" AT %IW2120 : Word;   // HAI def MW 266: actual water temperature magnet compressor unit 4 K26
   "DP_ATV_ERR_CODE_N9" AT %MW50 : Int;   // DP Slave +N9 (active cooling) activation error code
   "DP_ATV_TSK_RUN_N9" AT %M52.4 : Bool;   // DP Slave +N9 (active cooling) activation busy flag
   "HDO_LMP_BU_K2" AT %Q16.4 : Bool;   // HDO def M 136.4: Lamp blue +K2
   "HDO_LMP_BU_K8" AT %Q272.4 : Bool;   // HDO def M 160.4: Lamp blue +K8
   "HDO_LMP_BU_K9" AT %Q276.7 : Bool;   // HDO def M 165.7: Lamp blue +K9
   "HDO_LMP_GN_K2" AT %Q16.3 : Bool;   // HDO def M 136.3: Lamp green +K2
   "HDO_LMP_GN_K8" AT %Q272.3 : Bool;   // HDO def M 160.3: Lamp green +K8
   "HDO_LMP_GN_K9" AT %Q276.6 : Bool;   // HDO def M 165.6: Lamp green +K9
   "HDO_LMP_MAG_ACTIVE" AT %Q16.6 : Bool;   // HDO def M 136.6: Lamp magnet active( Lift+ Field on)
   "HDO_LMP_RD_K2" AT %Q16.1 : Bool;   // HDO def M 136.1: Lamp red +K2
   "HDO_LMP_RD_K8" AT %Q272.1 : Bool;   // HDO def M 160.1: Lamp red +K8
   "HDO_LMP_RD_K9" AT %Q276.4 : Bool;   // HDO def M 165.4: Lamp red +K9
   "HDI_LS_LO_XT_CLP_OP" AT %I276.5 : Bool;   // HDI def M 99.5: limit switch lower crystal clamp open
   "HDI_LS_LO_XT_CLP_PLATE" AT %I277.0 : Bool;   // HDI def M 100.0: limit switch upper crystal clamp plate
   "HDI_LS_LO_XT_CLP_SAVE" AT %I276.7 : Bool;   // HDI def M 99.7: limit switch lower crystal clamp save
   "HDI_LS_MAG_LFT_DN" AT %I34.3 : Bool;   // HDI def M 90.3: limit switch magnet lift down
   "HDO_XT_ROT_ENB" AT %Q272.5 : Bool;   // HDO def M 160.5: controller enable crystal rotation
   "HTR_1_AUX_DLY" AT %T72 : Timer;   // heater 1 auxiliary fault delay timer
   "HTR_1_TAS_DLY" AT %T70 : Timer;   // heater 1 temperature fault delay timer
   "HTR_1_WFS_DLY" AT %T71 : Timer;   // heater 1 waterflow fault delay timer
   "HTR_2_AUX_DLY" AT %T75 : Timer;   // heater 2 auxiliary fault delay timer
   "HTR_2_TAS_DLY" AT %T73 : Timer;   // heater 2 temperature fault delay timer
   "HTR_2_WFS_DLY" AT %T74 : Timer;   // heater 2 waterflow fault delay timer
   "HTR_AUX_DLY" AT %T94 : Timer;
   "HTR_TAS_DLY" AT %T92 : Timer;
   "HTR_WFS_DLY" AT %T93 : Timer;
   "P_STA_WTR_HTR" AT %IW2044 : Word;
   "P_STA_WTR_MAG_CAB" AT %IW2170 : Word;
   "P_STA_WTR_MAG_CO1" AT %IW2152 : Word;
   "P_STA_WTR_MAG_CO2" AT %IW2140 : Word;
   "P_STA_WTR_MAG_CO3" AT %IW2128 : Word;
   "P_STA_WTR_MAG_CO4" AT %IW2122 : Word;
   "P_STA_WTR_PWR_CAB" AT %IW2026 : Word;
   "P_STA_WTR_PWR_CAB2" AT %IW2032 : Word;
   "P_STA_WTR_SOC_BCH" AT %IW2176 : Word;
   "P_STA_WTR_TCH" AT %IW2092 : Word;
   "P_STA_WTR_TEC_FLG" AT %IW2116 : Word;
   "P_STA_WTR_UP_FCH" AT %IW2134 : Word;
   "P_STA_WTR_VPTS" AT %IW2080 : Word;
   "P_STA_WTR_XT_SFT" AT %IW2038 : Word;
   "BM_MCC_ON_TME" AT %T131 : Timer;   // melt contact control on time
   "HDI_FCH_APS" AT %I33.1 : Bool;   // HDI def M 89.1: pressure furnace chamber 1000 mbar
   "HDI_FCH_LFT_SDL_NUT" AT %I32.0 : Bool;   // HDI def M 88.0: safety limit switch furnace chamber lift spindle nut
   "HDI_FDR_APS" AT %I33.2 : Bool;   // HDI def M 89.2: pressure feeder 1000 mbar
   "HDI_FDR_HOP_CON" AT %M89.5 : Bool;   // HDI def M 89.5: hopper connected to feeder
   "HDI_FDR_LS_V3_2_CL" AT %I280.3 : Bool;   // HDI def M 103.3: Valve position V3_2 closed
   "HDI_FDR_LS_V3_2_OP" AT %I280.2 : Bool;   // HDI def M 103.2: valve position V3_2 open
   "HDI_FIL_2_APS" AT %I33.3 : Bool;   // HDI def M 89.3: atmospheric pressure filter 2
   "HDI_FIL_APS" AT %I18.4 : Bool;   // HDI def M 74.4: pressure filter 1000 mbar
   "HDI_FU_P2_RDY" AT %I144.0 : Bool;   // HDI def M 104.0: Frequency converter P2 ready/ no fault
   "HDI_GCH_APS" AT %I33.0 : Bool;   // HDI def M 89.0: pressure gate chamber 1000 mbar
   "HDI_KEY_XT_LFT_SRV" AT %I273.7 : Bool;   // HDI def M 96.7: Key switch service mode crystal lift
   "HDI_LSR_SEN_OBJ_DET" AT %I280.4 : Bool;   // HDI def M 103.4: spare digital input
   "HDI_LS_FCH_HOOK_HOME" AT %I32.3 : Bool;   // HDI def M 88.3: limit switch furnace chamber hook in home position
   "HDI_LS_FCH_HOOK_WORK" AT %I32.2 : Bool;   // HDI def M 88.2: limit switch furnace chamber hook in working position
   "P_reserve_3_X08_WTR_TMP" AT %IW2156 : Word;
   "P_reserve_4_X07_WTR_FLW" AT %IW2196 : Word;
   "P_reserve_4_X07_WTR_TMP" AT %IW2198 : Word;
   "P_reserve_4_X08_WTR_FLW" AT %IW2202 : Word;
   "P_reserve_4_X08_WTR_TMP" AT %IW2204 : Word;
   "P_reserve_STA_1_X07" AT %IW2056 : Word;
   "P_reserve_STA_1_X08" AT %IW2062 : Word;
   "P_reserve_STA_2_X06" AT %IW2098 : Word;
   "P_reserve_STA_2_X07" AT %IW2104 : Word;
   "P_reserve_STA_2_X08" AT %IW2110 : Word;
   "P_reserve_STA_3_X08" AT %IW2158 : Word;
   "P_reserve_STA_4_X07" AT %IW2200 : Word;
   "P_reserve_STA_4_X08" AT %IW2206 : Word;
   "HDI_P1_WD" AT %I18.3 : Bool;   // HDI def M 74.3: pump unit (P1) watchdog
   "HDI_P1_WRN" AT %I18.0 : Bool;   // HDI def M 74.0: pump unit (P1) warning
   "HDI_SLS_FCH_LFT" AT %I35.5 : Bool;   // HDI def M 91.5: Safety limit switch furnace chamber lift
   "HDI_SLS_GCH_LFT" AT %I272.6 : Bool;   // HDI def M 95.6: Safety limit switch gate chamber lift
   "HDI_SLS_MAG_LFT" AT %I34.4 : Bool;   // HDI def M 90.4: Safety limit switch magnet lift
   "HDI_SLS_TCH_LFT" AT %I279.4 : Bool;   // HDI def M 102.4: Safety limit switch top chamber lift
   "HDI_SLS_TEC_FLG_LFT" AT %I35.4 : Bool;   // HDI def M 91.4: Safety limit switch technolgy flange lift
   "HDI_SPARE_144_1" AT %I144.1 : Bool;   // HDI def M 104.1: spare digital input
   "HDI_SPARE_144_2" AT %I144.2 : Bool;   // HDI def M 104.2: spare digital input
   "HDI_SPARE_144_3" AT %I144.3 : Bool;   // HDI def M 104.3: spare digital input
   "HDI_SPARE_144_4" AT %I144.4 : Bool;   // HDI def M 104.4: spare digital input
   "HDI_SPARE_144_5" AT %I144.5 : Bool;   // HDI def M 104.5: spare digital input
   "HDI_SPARE_144_6" AT %I144.6 : Bool;   // HDI def M 104.6: spare digital input
   "HDI_SPARE_144_7" AT %I144.7 : Bool;   // HDI def M 104.7: spare digital input
   "HDI_SPARE_16_2" AT %I16.2 : Bool;   // HDI def M 72.4: spare digital input
   "HDI_SPARE_16_4" AT %I16.4 : Bool;   // HDI def M 72.4: spare digital input
   "HDO_LMP_YE_K2" AT %Q16.2 : Bool;   // HDO def M 136.2: Lamp yellow +K2
   "HDO_LMP_YE_K8" AT %Q272.2 : Bool;   // HDO def M 160.2: Lamp yellow +K8
   "HDO_LMP_YE_K9" AT %Q276.5 : Bool;   // HDO def M 165.5: Lamp yellow +K9
   "HDO_LO_FCH_SW_BRK" AT %Q96.3 : Bool;   // HDO def M 150.3: Valve block lower chamber swivel release brake
   "HDO_LSR_SEN_PWR_ON" AT %Q273.2 : Bool;   // HDO def M 161.2: supply voltage for laser sensor on
   "HDO_MAG_LFT_DN" AT %Q33.3 : Bool;   // HDO def M 143.3: Magnet lift drive downwards
   "PFM_PRESET_VSL_SW" AT %M39.0 : Bool;
   "PFM_TEC_FLG_DN" AT %M38.0 : Bool;
   "P_BM_ACT_WTR_FLW_GCH_H" AT %IW2064 : Word;   // HAI def MW 271: actual water flow gate chamber valve housing K04
   "P_BM_ACT_WTR_FLW_GCH_V" AT %IW2070 : Word;   // HAI def MW 280: actual water flow gate chamber valve K05
   "P_BM_ACT_WTR_FLW_HTR" AT %IW2040 : Word;   // HAI def MW 253: actual water flow heater power supply K20
   "P_BM_ACT_WTR_FLW_MAG_CAB" AT %IW2166 : Word;   // HAI def MW 318: actual water flow magnet power supply K30
   "P_BM_ACT_WTR_FLW_MAG_CO1" AT %IW2148 : Word;   // HAI def MW 282: actual water flow magnet compressor unit 1 K29
   "P_BM_ACT_WTR_FLW_MAG_CO2" AT %IW2136 : Word;   // HAI def MW 291: actual water flow magnet compressor unit 2 K28
   "P_BM_ACT_WTR_FLW_MAG_CO3" AT %IW2124 : Word;   // HAI def MW 255: actual water flow magnet compressor unit 3 K27
   "P_BM_ACT_WTR_FLW_MAG_CO4" AT %IW2118 : Word;   // HAI def MW 264: actual water flow magnet compressor unit 4 K26
   "P_BM_ACT_WTR_FLW_PWR_CAB" AT %IW2022 : Word;   // HAI def MW 354: actual water flow high current cables Main K18
   "P_BM_ACT_WTR_FLW_PWR_CAB2" AT %IW2028 : Word;   // HAI def MW 345: actual water flow high current cables Bot K19
   "P_BM_ACT_WTR_FLW_SOC_BCH" AT %IW2172 : Word;   // HAI def MW 327: actual water flow socket bottom chamber K13
   "P_BM_ACT_WTR_FLW_TCH" AT %IW2088 : Word;   // HAI def MW 237: actual water flow top chamber K07
   "P_BM_ACT_WTR_FLW_TEC_FLG" AT %IW2112 : Word;   // HAI def MW 273: actual water flow technolity chamber K08
   "P_BM_ACT_WTR_FLW_UP_FCH" AT %IW2130 : Word;   // HAI def MW 336: actual water flow upper furnace chamber K10
   "P_BM_ACT_WTR_FLW_VPTS" AT %IW2076 : Word;   // HAI def MW 289: actual water flow view ports K06
   "P_BM_ACT_WTR_FLW_XT_SFT" AT %IW2034 : Word;   // HAI def MW 244: actual water flow seed shaft K02
   "HDO_FDR_V11_CL" AT %Q225.7 : Bool;   // HDO def M 151.7: Valve block close V11 (isolation valve feeder)
   "HDO_FDR_V11_CVR_CL" AT %Q226.1 : Bool;   // HDO def M 152.1: Valve block close cover V11 (isolation valve feeder)
   "HDO_FDR_V11_CVR_OP" AT %Q226.0 : Bool;   // HDO def M 152.0: Valve block open cover V11 (isolation valve feeder)
   "HDO_FDR_V11_OP" AT %Q225.6 : Bool;   // HDO def M 151.6: Valve block open V11 (isolation valve feeder)
   "HDO_FU_FCB_HDL_ON" AT %Q32.7 : Bool;   // HDO def M 142.7: Frequency converter FCB handling on
   "HDO_FU_GCB_HDL_ON" AT %Q273.1 : Bool;   // HDO def M 161.1: Frequency converter GCB handling on
   "HDO_GCH_LFT_ENB" AT %Q274.7 : Bool;   // HDO def M 163.7: controller enable gate chamber lift
   "HDO_GCH_SW_LOCK" AT %Q225.2 : Bool;   // HDO def M 151.2: Valve block gate chamber swivel lock close
   "HDO_GCH_SW_UNLOCK" AT %Q225.3 : Bool;   // HDO def M 151.3: Valve block gate chamber swivel lock open
   "HDO_GTE_V_LFT_ENB" AT %Q276.0 : Bool;   // HDO def M 165.0: controller enable gate valve lift
   "HDO_GTE_V_SW_ENB" AT %Q276.1 : Bool;   // HDO def M 165.1: controller enable gate valve swivel
   "HDO_HOR_MAG_ACTIVE" AT %Q16.5 : Bool;   // HDO def M 136.5: Horn magnet active( Lift)
   "HDI_LS_UP_XT_CLP_CL" AT %I276.1 : Bool;   // HDI def M 99.1: limit switch upper crystal clamp closed
   "HDI_LS_UP_XT_CLP_FLT" AT %I275.6 : Bool;   // HDI def M 98.6: limit switch upper crystal clamp fault
   "HDI_LS_UP_XT_CLP_OP" AT %I276.0 : Bool;   // HDI def M 99.0: limit switch upper crystal clamp open
   "HDI_LS_UP_XT_CLP_PLATE" AT %I276.3 : Bool;   // HDI def M 99.3: limit switch upper crystal clamp plate
   "HDI_LS_UP_XT_CLP_SAVE" AT %I276.2 : Bool;   // HDI def M 99.2: limit switch upper crystal clamp save
   "HDI_LS_V11_CL" AT %M89.4 : Bool;   // HDI def M 89.4: V 11 closed (isolation valve feeder)
   "SysCycle100ms" AT %M2.0 : Bool;   // System Cycle: 100 ms
   "SysCycle1_6s" AT %M2.6 : Bool;   // System Cycle: 1600 ms
   "SysCycle1s" AT %M2.5 : Bool;   // System Cycle: 1000 ms
   "SysCycle200ms" AT %M2.1 : Bool;   // System Cycle: 200 ms
   "SysCycle2s" AT %M2.7 : Bool;   // System Cycle: 2000 ms
   "SysCycle400ms" AT %M2.2 : Bool;   // System Cycle: 400 ms
   "SysCycle500ms" AT %M2.3 : Bool;   // System Cycle: 500 ms
   "SysCycle800ms" AT %M2.4 : Bool;   // System Cycle: 800 ms
   "SysEdgeFlag100ms" AT %M3.0 : Bool;   // System Cycle: Edge Flag 100 ms
   "SysEdgeFlag1_6s" AT %M4.4 : Bool;   // System Cycle: Edge Flag 1600 ms
   "SysEdgeFlag1s" AT %M4.2 : Bool;   // System Cycle: Edge Flag 1000 ms
   "SysEdgeFlag200ms" AT %M3.2 : Bool;   // System Cycle: Edge Flag 200 ms
   "SysEdgeFlag2s" AT %M4.6 : Bool;   // System Cycle: Edge Flag 2000 ms
   "P_BM_PWR_SPL_1_ACT_CUR" AT %ID918 : Real;   // actual current heater 1
   "P_BM_PWR_SPL_1_ACT_PWR" AT %ID914 : Real;   // actual power heater 1
   "P_BM_PWR_SPL_1_ACT_RESIS" AT %ID922 : Real;   // resistance heater 1
   "P_BM_PWR_SPL_1_ACT_VLT" AT %ID910 : Real;   // actual voltage heater 1
   "P_BM_PWR_SPL_1_BUS_MINUS" AT %ID930 : Real;   // bus minus heater 1
   "P_BM_PWR_SPL_1_BUS_PLUS" AT %ID926 : Real;   // bus plus heater 1
   "P_BM_PWR_SPL_1_SET_PWR" AT %QD898 : Real;   // setpoint power heater 1
   "P_BM_PWR_SPL_2_ACT_CUR" AT %ID942 : Real;   // actual current heater 2
   "P_BM_PWR_SPL_2_ACT_PWR" AT %ID938 : Real;   // actual power heater 2
   "P_BM_PWR_SPL_2_ACT_RESIS" AT %ID946 : Real;   // resistance heater 2
   "P_BM_PWR_SPL_2_ACT_VLT" AT %ID934 : Real;   // actual voltage heater 2
   "P_BM_PWR_SPL_2_BUS_MINUS" AT %ID954 : Real;   // bus minus heater 2
   "P_BM_PWR_SPL_2_BUS_PLUS" AT %ID950 : Real;   // bus plus heater 2
   "HDI_LS_GCH_BEL_UP" AT %I274.6 : Bool;   // HDI def M 97.6: limit switch gate chamber bellow in upper position
   "HDI_LS_GCH_DN" AT %I272.1 : Bool;   // HDI def M 95.1: limit switch gate chamber in lower position
   "HDI_LS_GCH_DOOR_CL" AT %I278.7 : Bool;   // HDI def M 101.7: limit switch gate chamber door closed
   "HDI_LS_GCH_DOOR_OP" AT %I278.6 : Bool;   // HDI def M 101.6: limit switch gate chamber door opened
   "HDI_LS_GCH_SW_CLN" AT %I272.3 : Bool;   // HDI def M 95.3: limit switch gate chamber swivelled in cleaning pos
   "HDI_LS_GCH_SW_IN" AT %I272.2 : Bool;   // HDI def M 95.2: limit switch gate chamber swivelled in
   "HDI_LS_GCH_SW_LOCK" AT %I272.5 : Bool;   // HDI def M 95.5: limit switch gate chamber swivel locked
   "HDI_LS_GCH_SW_OUT" AT %I272.4 : Bool;   // HDI def M 95.4: limit switch gate chamber swivelled out
   "HDI_LS_GCH_UP" AT %I272.0 : Bool;   // HDI def M 95.0: limit switch gate chamber in upper position
   "HDI_LS_HOI_TOOL_INST" AT %I277.1 : Bool;   // HDI def M 100.1: limit switch HOI tool installed
   "HDI_LS_LO_XT_CLP_CL" AT %I276.6 : Bool;   // HDI def M 99.6: limit switch lower crystal clamp closed
   "HDI_LS_LO_XT_CLP_FLT" AT %I276.4 : Bool;   // HDI def M 99.4: limit switch lower crystal clamp fault
   "HDO_SPARE_32_3" AT %Q32.3 : Bool;   // HDO def M 142.3: spare digital output
   "HDO_SPARE_32_4" AT %Q32.4 : Bool;   // HDO def M 142.4: spare digital output
   "HDO_SPARE_33_5" AT %Q33.5 : Bool;   // HDO def M 143.5: spare digital output
   "HDO_SPARE_33_6" AT %Q33.6 : Bool;   // HDO def M 143.6: spare digital output
   "HDO_SPARE_33_7" AT %Q33.7 : Bool;   // HDO def M 143.7: spare digital output
   "HDO_SPARE_34_2" AT %Q34.2 : Bool;   // HDO def M 144.2: spare digital output
   "HDO_SPARE_34_3" AT %Q34.3 : Bool;   // HDO def M 144.3: spare digital output
   "HDO_SPARE_34_4" AT %Q34.4 : Bool;   // HDO def M 144.4: spare digital output
   "HDO_SPARE_34_5" AT %Q34.5 : Bool;   // HDO def M 144.5: spare digital output
   "HDO_SPARE_34_6" AT %Q34.6 : Bool;   // HDO def M 144.6: spare digital output
   "HDO_SPARE_34_7" AT %Q34.7 : Bool;   // HDO def M 144.7: spare digital output
   "HDO_TCH_LFT_ENB" AT %Q275.6 : Bool;   // HDO def M 164.6: controller enable top chamber lift
   "P_BM_ETH_FLT_MON_IIST1" AT %IW1058 : Int;   // Main heater earth fault monitoring voltage out
   "P_BM_ETH_FLT_MON_IIST2" AT %IW1063 : Int;   // Bottom heater earth fault monitoring voltage out
   "P_BM_ETH_FLT_MON_UIST1" AT %IW1056 : Int;   // Main heater earth fault monitoring voltage in
   "FLT_OUT_OF_MELT_DLY" AT %T133 : Timer;   // delay timer out of melt fault
   "FL_FDG_RTE_OFF" AT %M5.7 : Bool;   // Flange Regelung Feed rate aus
   "P_HAI_ACC_SPARE_11" AT %IW780 : Word;   // HAI def MW 268: ACC spare
   "P_HAI_ACC_SPARE_810" AT %IW810 : Word;   // HAI def MW 268: ACC spare
   "P_HAI_ACC_WTR_FLW_IN" AT %IW806 : Word;   // HAI def MW 264: ACC waterflow input
   "P_HAI_ACC_WTR_FLW_OUT" AT %IW804 : Word;   // HAI def MW 262: ACC waterflow output
   "P_HAI_ACC_WTR_PRS_IN" AT %IW802 : Word;   // HAI def MW 260: ACC water pressure
   "HDO_SPARE_144_7" AT %Q144.7 : Bool;   // HDO def M 152.7: spare digital output
   "HDO_SPARE_16_7" AT %Q16.7 : Bool;   // HDO def M 136.7: spare digital output
   "HDO_SPARE_18_0" AT %Q18.0 : Bool;   // HDO def M 138.0: spare digital output
   "HDO_SPARE_18_1" AT %Q18.1 : Bool;   // HDO def M 138.1: spare digital output
   "HDO_SPARE_18_2" AT %Q18.2 : Bool;   // HDO def M 138.2: spare digital output
   "HDO_SPARE_18_3" AT %Q18.3 : Bool;   // HDO def M 138.3: spare digital output
END_VAR

TYPE "UDT_ANY_POINTER"
VERSION : 0.0
   STRUCT
      Syntax_Id : Byte;   // MUST always be 10 Hex !!
      DataType : Byte;   // code for data type e.g. 01=BOOL, 02=BYTE....
      Count : Word;   // number of bytes
      DB_Number : Word;   // number of DB
      Byte_Pointer : DWord;   // pointer to bit and byte adress
   END_STRUCT;
END_TYPE

TYPE "UDT_DRV_DAT_IN_i550"
VERSION : 0.0
   STRUCT
      STATW : Word;
      ACT_Speed_Hz_0_1 : Word;
      ACT_Current : Word;
      Error_code : Word;
   END_STRUCT;
END_TYPE

TYPE "UDT_DRV_DAT_OUT_i550"
VERSION : 0.0
   STRUCT
      CTRW : Word;
      SET_Speed_Hz_0_1 : Word;
      W_Bit_out_spare : Word;
   END_STRUCT;
END_TYPE

TYPE "UDT_DRV_LENZE_i550"
VERSION : 0.0
   STRUCT
      Input : "UDT_DRV_DAT_IN_i550";
      Output : "UDT_DRV_DAT_OUT_i550";
   END_STRUCT;
END_TYPE

TYPE "UDT_DRV_DAT_OUT_BOOL"
VERSION : 0.0
   STRUCT
      Spare_7 : Bool;
      Spare_8 : Bool;
      Spare_9 : Bool;
      Spare_10 : Bool;
      Enab_ext_pos : Bool;
      Enab_ext_vel : Bool;
      Enab_ext_acc_dcc_jerk : Bool;
      Enab_ext_torque_limit : Bool;
      Profile_BIT_0 : Bool;   // Profile is choosen out of the 4 Bits 0001 = Profile 1 // 0101 = Profile 5
      Profile_BIT_1 : Bool;
      Profile_BIT_2 : Bool;
      Profile_BIT_3 : Bool;
      Do_pos_drv : Bool;
      Abort_pos_drv : Bool;
      Continue_pos_drv : Bool;
      Touch_probe_acti : Bool;
      Stop : Bool;
      Start_homing : Bool;
      Reset_ref_pos : Bool;
      Spare_4 : Bool;
      Spare_5 : Bool;
      Act_ext_vel_over : Bool;
      Disable_Break : Bool;
      Spare_6 : Bool;
      Spare_1 : Bool;
      Spare_2 : Bool;
      Activate_quick_stop : Bool;
      Enable : Bool;
      Spare_3 : Bool;
      Jog_pos : Bool;
      Jog_neg : Bool;
      Res_error : Bool;
   END_STRUCT;
END_TYPE

TYPE "UDT_DRV_DAT_OUT_PARA"
VERSION : 0.0
   STRUCT
      Ext_vel_over : DWord;   // 0.00 .. 100.00%
      Ext_vel : DWord;   // 4 Nachkomma
      Ext_pos : DWord;   // 4 Nachkomma
      Ext_acc : DWord;   // 4 Nachkomma
      Ext_dcc : DWord;   // 4 Nachkomma
      Ext_jerk : DWord;   // 2 Nachkomma
      Ext_torq_lim : DWord;   // 2 Nachkomma 0.00 - 200.00%
   END_STRUCT;
END_TYPE

TYPE "UDT_DRV_DAT_OUT"
VERSION : 0.0
   STRUCT
      Control_Bools : "UDT_DRV_DAT_OUT_BOOL";
      Control_Para : "UDT_DRV_DAT_OUT_PARA";
   END_STRUCT;
END_TYPE

TYPE "UDT_DRV_DAT_IN_BOOL_1"
VERSION : 0.0
   STRUCT
      Touch_probe_home : Bool;
      Spare_5 : Bool;
      Spare_6 : Bool;
      Spare_7 : Bool;
      Ext_pos_active : Bool;
      Ext_vel_active : Bool;
      Ext_acc_dec_jer_active : Bool;
      Ext_torq_lim_active : Bool;
      Profile_BIT_0 : Bool;
      Profile_BIT_1 : Bool;
      Profile_BIT_2 : Bool;
      Profile_BIT_3 : Bool;
      Pos_cont_active : Bool;
      Pos_cont_done : Bool;
      LS_neg : Bool;
      LS_pos : Bool;
      Halt_active : Bool;
      Spare_3 : Bool;
      Set_pos_reached : Bool;
      Spare_4 : Bool;
      Standstill : Bool;
      Dir_inv : Bool;
      Brake_released : Bool;
      STO_active : Bool;
      Drv_ready : Bool;
      Homing_active : Bool;
      Op_enabled : Bool;
      Drv_error : Bool;
      Homing_finished : Bool;
      Qsp_active : Bool;
      Jog_active : Bool;
      Drv_waring : Bool;
   END_STRUCT;
END_TYPE

TYPE "UDT_DRV_DAT_IN_BOOL_2"
VERSION : 0.0
   STRUCT
      Spare_1 : Bool;
      Spare_2 : Bool;
      Spare_3 : Bool;
      Spare_4 : Bool;
      Spare_5 : Bool;
      Spare_6 : Bool;
      Spare_7 : Bool;
      Spare_8 : Bool;
      Spare_9 : Bool;
      Spare_10 : Bool;
      Spare_11 : Bool;
      Spare_12 : Bool;
      Spare_13 : Bool;
      Spare_14 : Bool;
      Spare_15 : Bool;
      Spare_16 : Bool;
      Safe_dir_pos : Bool;
      Safe_dir_neg : Bool;
      Safe_lim_inc : Bool;
      Safe_stp_emg : Bool;
      ES_active : Bool;
      Op_mod_sel : Bool;
      Spare_17 : Bool;
      Spare_18 : Bool;
      Safe_torq_off : Bool;
      Safe_stp_1 : Bool;
      Safe_stp_2 : Bool;
      Safe_op_stp : Bool;
      Safely_lim_vel_1 : Bool;
      Safely_lim_vel_2 : Bool;
      Safely_lim_vel_3 : Bool;
      Safely_lim_vel_4 : Bool;
   END_STRUCT;
END_TYPE

TYPE "PAR_DATA"
VERSION : 0.0
   STRUCT
      PAR : Array[1..10, 1..21] of Real;
   END_STRUCT;
END_TYPE

TYPE "UDT_DRV_DAT_IN_PARA"
VERSION : 0.0
   STRUCT
      Act_vel : DWord;   // 4 Nachkomma
      Act_pos : DWord;
      Error_code : DWord;   // Aktuelle Fehlernummer
      Act_torq : DWord;   // 2 Nachkomma
      Mon_sig : DWord;
      Spare_1 : DWord;
   END_STRUCT;
END_TYPE

TYPE "UDT_DRV_DAT_IN"
VERSION : 0.0
   STRUCT
      Status_Bools_1 : "UDT_DRV_DAT_IN_BOOL_1";
      Status_Bools_2 : "UDT_DRV_DAT_IN_BOOL_2";
      Status_Para : "UDT_DRV_DAT_IN_PARA";
   END_STRUCT;
END_TYPE

TYPE "UDT_DRV_LENZE_i950"
VERSION : 0.0
   STRUCT
      Input : "UDT_DRV_DAT_IN";
      Output : "UDT_DRV_DAT_OUT";
   END_STRUCT;
END_TYPE

DATA_BLOCK "SY"   // DB2
{ S7_Optimized_Access := 'FALSE' }
VERSION : 0.0
// --------------------------------------------------------------------------------
//     program     :    SY
//     description :    define all SY values       
//     name        :    G. Eibelsh鋟ser
//     date        :    28.10.99
// 
//     revision    : 
//     name        : 
//     date        :   
//     
//                     (c)PVA TePla AG       
//     --------------------------------------------------------------------------------
   VAR
      SIM_ON : Bool;   // simulation mode active
      SRM_ON : Bool;   // service mode active
      CTL_DIA_SMI : Bool;
      CTL_PRS_SMI : Bool;
      CTL_HTR_1_SMI : Bool;
      CTL_HTR_2_SMI : Bool;
      CTL_HTR_3_SMI : Bool;
      CTL_MAG_1_SMI : Bool;
      CTL_MAG_2_SMI : Bool;
      CTL_MLT_LVL_SMI : Bool;
      CTL_XT_ROT_SMI : Bool;
      CTL_CR_SPD_SMI : Bool;
      CTL_CR_ROT_SMI : Bool;
      CTL_GAS_FLOW_SMI : Bool;
      CTL_SI_FDR_SMI : Bool;
      CTL_DOP_FDR_SMI : Bool;
      CTL_DIA_ON : Bool;
      CTL_PRS_ON : Bool;
      CTL_HTR_1_ON : Bool;
      CTL_HTR_2_ON : Bool;
      CTL_MLT_LVL_ON : Bool;
      CTL_AVG_SPD_ON : Bool;
      CTL_AVG_CRUC_ROT_ON : Bool;
      CTL_MLT_TMP_ON : Bool;
      CTL_GRW_RTE_ON : Bool;
      CTL_CR_SPD_COF_SMI : Bool;
      CTL_MLT_DRIFT_ON : Bool;
      CTL_DIA_TMP_ON : Bool;
      CTL_GAP_ON : Bool;   // gap controller on
      CTL_AVG_OFFS_ON : Bool;   // offset controller on
      CTL_OFFS_SPEED_ON : Bool;
      CTL_GAP_SMI : Bool;
      DEVICE : Array[1..49] of Struct
         STATUS : Int;   // device status 0 = not init, 1 = ok, 2 = init error, 3 = fault, 9 = not active
         ENABLE : Bool;   // device is controled by plc via l2-bus
         ERROR_INDEX : Int;   // error index e.g. parameter no (see device manual)
         ERROR_CODE : DWord;   // error code e.g. error number (see device manual)
      END_STRUCT;
      RUN_TIME : DInt;
      OB1_PREV_CYCLE : Int;
      OB1_MIN_CYCLE : Int;
      OB1_MAX_CYCLE : Int;
   END_VAR
BEGIN
END_DATA_BLOCK

DATA_BLOCK "SW"   // DB3
{ S7_Optimized_Access := 'FALSE' }
VERSION : 0.0
// --------------------------------------------------------------------------------
//     program     :    SW
//     description :    software information      
//     name        :    L. Vogel
//     date        :    08.09.2018
// 
//     revision    :
//     name        :
//     date        :    
//                     (c)PVA GCS GmbH
//     --------------------------------------------------------------------------------
   VAR
      ACT_PLC_VERSION : Real := 2.13;
      ACT_PLC_CONFIG : Real := 40.0;
   END_VAR
BEGIN
END_DATA_BLOCK

DATA_BLOCK "PAR_SUB"   // DB9
{ S7_Optimized_Access := 'FALSE' }
VERSION : 0.0
// --------------------------------------------------------------------------------
//     program     :    PAR_SUB
//     description :    define all CONTROL parameter on sub pages         
//     name        :    G. Eibelsh鋟ser
//     date        :    22.01.2001
// 
//     revision    :
//     name        :
//     date        :    
//                     (c)CGS
//     --------------------------------------------------------------------------------
   VAR
      PRS_RP_MAX_DEV : Real;   // word 0
      PRS_RP_START : Real;
      PRS_RP_GRAD : Real;
      DIA_RP_MAX_DEV : Real;
      DIA_RP_START : Real;
      DIA_RP_GRAD : Real;
      HTR_1_TMP_RP_MAX_DEV : Real;
      HTR_1_TMP_RP_START : Real;
      HTR_1_TMP_RP_GRAD : Real;   // word 32
      HTR_2_TMP_RP_MAX_DEV : Real;
      HTR_2_TMP_RP_START : Real;
      HTR_2_TMP_RP_GRAD : Real;
      AV_PULL_SPD_RP_MAX_DEV : Real;
      AV_PULL_SPD_RP_START : Real;
      AV_PULL_SPD_RP_GRAD : Real;
      AV_CRUC_ROT_RP_MAX_DEV : Real;
      AV_CRUC_ROT_RP_START : Real;   // word 64
      AV_CRUC_ROT_RP_GRAD : Real;
      MELT_TMP_RP_MAX_DEV : Real;
      MELT_TMP_RP_START : Real;
      MELT_TMP_RP_GRAD : Real;
      GRO_RP_MAX_DEV : Real;
      GRO_RP_START : Real;
      GRO_RP_GRAD : Real;
      MLT_LVL_RP_MAX_DEV : Real;   // word 96
      MLT_LVL_RP_START : Real;
      MLT_LVL_RP_GRAD : Real;
      WRN_DST_UPR_CR_POS_LIM : Real;
      ALM_DST_UPR_CR_POS_LIM : Real;
      SPARE_116 : Real;
      FI_MOB_FDR_VIB : Real;
      FI_GRO_NE : Real;
      FI_TMP_HTR_1 : Real;   // word 128
      FI_TMP_HTR_2 : Real;
      FI_DIA_NE_T1 : Real;
      FI_DIA_SH_T1 : Real;
      FI_DIA_BY_T1 : Real;
      FI_GRO_SH : Real;
      FI_AV_SPD : Real;
      FI_MLT_LVL : Real;
      FI_AV_TMP_1 : Real;   // word 160
      FI_AV_TMP_2 : Real;
      FI_MLT_TMP_1 : Real;
      FI_MLT_TMP_2 : Real;
      FI_SH_AV_CRUC_ROT : Real;
      FI_BY_AV_CRUC_ROT : Real;
      FI_DIA_NE_T2 : Real;
      FI_DIA_SH_T2 : Real;
      FI_DIA_BY_T2 : Real;   // word 192
      FI_DIA_DYN_WIN_T1 : Real;
      FI_DIA_DYN_WIN_RR : Real;
      ACT_XT_WGT_DLY_T1 : Real;
      ME_V1_LWR_POS_LIM : Real;
      ME_V1_UPR_POS_LIM : Real;
      DI_V1_LWR_POS_LIM : Real;
      DI_V1_UPR_POS_LIM : Real;
      NE_V1_LWR_POS_LIM : Real;   // word 224
      NE_V1_UPR_POS_LIM : Real;
      SH_V1_LWR_POS_LIM : Real;
      SH_V1_UPR_POS_LIM : Real;
      BY_V1_LWR_POS_LIM : Real;
      BY_V1_UPR_POS_LIM : Real;
      RC_V1_LWR_POS_LIM : Real;
      RC_V1_UPR_POS_LIM : Real;
      EC_V1_LWR_POS_LIM : Real;   // word 256
      EC_V1_UPR_POS_LIM : Real;
      SD_V1_LWR_POS_LIM : Real;
      SD_V1_UPR_POS_LIM : Real;
      SCAM_MLT_LVL_T1 : Real;
      CTR_X_SCAM_2_ADJ : Real;
      CTR_Y_SCAM_2_ADJ : Real;
      FIL_CHG_V1_POS : Real;
      SPARE_288 : Real;   // word 288
      CAM_FLT_XT_ROT_STP : Real;
      CAM_FLT_CR_ROT_STP : Real;
      CAM_FLT_CR_LFT_DN : Real;
      CONE_TMP_HI_HTR_OFF : Real;
      CONE_TMP_HI_XT_ROT_STP : Real;
      CONE_TMP_HI_CR_ROT_STP : Real;
      CONE_TMP_HI_CR_LFT_DN : Real;
      CONE_FLW_LO_HTR_OFF : Real;   // word 320
      CONE_FLW_LO_XT_ROT_STP : Real;
      CONE_FLW_LO_CR_ROT_STP : Real;
      CONE_FLW_LO_CR_LFT_DN : Real;
      FNC_PRS_HI_HTR_OFF : Real;
      FNC_PRS_HI_XT_ROT_STP : Real;
      FNC_PRS_HI_CR_ROT_STP : Real;
      FNC_PRS_HI_CR_LFT_DN : Real;
      XT_WGT_CHG_HTR_OFF : Real;   // word 352
      XT_WGT_CHG_XT_ROT_STP : Real;
      XT_WGT_CHG_CR_ROT_STP : Real;
      SPARE_364 : Real;
      SPARE_368 : Real;
      SPARE_372 : Real;
      SPARE_376 : Real;
      XT_DIA_CHG_CR_LFT_DN : Real;
      WTR_FLW_CONE_LO_LIM : Real;   // word 384
      WTR_TMP_CONE_HI_LIM : Real;
      PRS_ABV_UPR_LIM : Real;
      XT_WGT_CHG_ABV_UPR_LIM : Real;
      XT_WGT_CHG_BLW_LWR_LIM : Real;
      XT_DIA_CHG_ABV_UPR_LIM : Real;
      XT_DIA_CHG_BLW_LWR_LIM : Real;
      SPARE_412 : Real;
      SET_HTR_1_RES : Real;   // word 416
      HTR_1_UPR_RES_RNG : Real;
      HTR_1_LWR_RES_RNG : Real;
      SET_HTR_2_RES : Real;
      HTR_2_UPR_RES_RNG : Real;
      HTR_2_LWR_RES_RNG : Real;
      RES_DEV_CNT_DLY : Real;
      SPARE_444 : Real;
   END_VAR
BEGIN
END_DATA_BLOCK

DATA_BLOCK "PAR_MAIN"   // DB10
{ S7_Optimized_Access := 'FALSE' }
VERSION : 0.0
// --------------------------------------------------------------------------------
//     program     :    PAR_MAIN
//     description :    define all main process parameter        
//     name        :    K. Kalkowski
//     date        :    28.10.99
// 
//     revision    :
//     name        :
//     date        :    
//                     (c)LEYBOLD SYSTEMS
//     --------------------------------------------------------------------------------
   VAR
      CH_QRZ_WALL_THICKN : Real;   // dword 0
      CH_QRZ_BOTTOM_THICKN : Real;
      CH_GRAPH_TRANS_RAD : Real;
      CH_GRAPH_BOTTOM_RAD : Real;
      CH_GRAPH_INNER_DIA : Real;
      CH_DIST_BOTTOM_SHAFT : Real;
      CH_SILICON_CHARGE : Real;
      PD_AMT_PRG_CYC : Real;
      PD_PRG_INLET_V5 : Real;   // dword 32
      PD_PRG_GAS_FLW : Real;
      PD_PRG_TME : Real;
      PD_PRG_STR_PRS : Real;
      PD_10_MBAR_TME : Real;
      PD_1_MBAR_TME : Real;
      PD_01_MBAR_TME : Real;
      PD_005_MBAR_TME : Real;
      PD_FINAL_PRS : Real;   // dword 64
      PD_LEAKTEST_TME : Real;
      PD_MAX_LEAKRATE : Real;
      PD_XT_ROT : Real;
      PD_CR_ROT : Real;
      PD_SOFTPUMP_DELAY : Real;
      ME_FDR_MAX_LRT : Real;
      ME_FDR_FINAL_PRS : Real;
      ME_FDR_FLP_TME_OP : Real;   // dword 96
      ME_FDR_FLP_TME_CL : Real;
      ME_FDR_STEP : Real;
      ME_DETECT_STEP : Real;
      ME_LSR_STEP : Real;
      ME_HI_CR_POS_REF_LVL : Real;
      ME_CR_POS_ABV_REF_LVL : Real;
      ME_FDR_LEAK_TST_TME : Real;
      ME_FDR_MAX_PRS_DROP : Real;   // dword 128
      DI_TMP_DEV_START : Real;
      DI_TMP_DIPPING : Real;
      DI_TMP_DEV_DIP : Real;
      DI_MIN_TME : Real;
      DI_TMP_GAP_HTR_1 : Real;
      DI_TMP_GAP_HTR_2 : Real;
      DI_TMP_DEC_HTR_1 : Real;
      DI_TMP_DEC_HTR_2 : Real;   // dword 160
      DI_INI_PWR_1 : Real;
      DI_INI_PWR_2 : Real;
      DI_AUTO_THR_ADJ : Real;
      ME_AMT_OF_FDG_STP : Real;
      NE_XT_SPD_INC : Real;
      NE_DIA : Real;
      NE_LEN : Real;
      NE_MLT_CONTACT_CTL : Real;   // dword 192
      DIA_MSR_PRD_NE : Real;
      NE_MIN_DIA : Real;
      SH_MLT_CONTACT_CTL : Real;
      SH_BODY_TRANS_GRW : Real;
      SH_BODY_TRANS_DLY_TME : Real;
      SH_TMP_GAP_HTR_1 : Real;
      SH_TMP_GAP_HTR_2 : Real;
      SH_BODY_TRANS_DIA : Real;   // dword 224
      SH_BODY_TRANS_SPD : Real;
      SH_BODY_START_DIA : Real;
      SH_CRUC_ROT_CTL_ON : Real;
      SH_START_CRUC_ROT : Real;
      SH_LSR_LVL_CTL_ON : Real;
      DIA_MSR_PRD_SH : Real;
      DIA_MSR_PRD_BY : Real;
      BY_XT_DIA : Real;   // dword 256
      BY_XT_LEN : Real;
      BY_CRUC_ROT_CTL_ON : Real;
      BY_CRUC_ROT_OFFS_RP_GRAD : Real;
      BY2_LEN_RP_START : Real;
      BY2_RP_TME : Real;
      BY_LSR_LVL_CTL_ON : Real;
      EC_XT_LEN : Real;
      EC_MLT_CONTACT_CTL : Real;   // dword 288
      EC_ROT_ABS_INC : Real;
      BY_MLT_CONTACT_CTL : Real;
      EC_V21_TI_TILL_OPEN : Real;
      EC_V21_OPEN_TIME : Real;
      ME_STEP_MLT_LVL_CHECK : Real;
      BY_CTL_MLT_DRIFT_ON : Real;
      BY_XT_LGH_MLT_LVL_RST : Real;
      SD_TME_TILL_VENT : Real;   // dword 320
      SD_TME_DUST_SEP : Real;
      SD_FLW_DUST_SEP : Real;
      SD_VALVE_DUST_SEP : Real;
      SD_LEAKTEST_TME : Real;
      SD_MAX_LEAKRATE : Real;
      SD_FINAL_PRS : Real;
      SD_V21_TI_TILL_OPEN : Real;
      SD_V21_OPEN_TIME : Real;   // dword 352
      RC_AMT_PRG_CYC : Real;
      RC_PRG_INLET_V5 : Real;
      RC_PRG_GAS_FLW : Real;
      RC_XT_ROT : Real;
      RC_CR_ROT : Real;
      RC_XT_POS : Real;
      RC_CR_POS : Real;
      RC_HTR_1_INC : Real;   // dword 384
      RC_HTR_2_INC : Real;
      RC_GAS_1_FLW : Real;
      RC_GAS_2_FLW : Real;
      RC_PRS : Real;
      RC_MAG_AV_CUR : Real;
      RC_MAG_RATIO_CUR : Real;
      RC_PRG_TME : Real;
      RC_PRG_STR_PRS : Real;   // dword 416
      BY_DIA_CTRL_ON_DLY : Real;
      ME_FDR_PUR_CYC : Real;
      PD_WAIT_TME_FIN_PRS : Real;
      CTL_HTR_1_TMP_GN_DIP : Real;
      CTL_HTR_1_TMP_TI_DIP : Real;
      CTL_HTR_1_TMP_TD_DIP : Real;
      CTL_HTR_1_TMP_T1_DIP : Real;
      CTL_HTR_1_TMP_GN : Real;   // dword 448
      CTL_HTR_1_TMP_TI : Real;
      CTL_HTR_1_TMP_TD : Real;
      CTL_HTR_1_TMP_T1 : Real;
      CTL_HTR_2_TMP_GN_DIP : Real;
      CTL_HTR_2_TMP_TI_DIP : Real;
      CTL_HTR_2_TMP_TD_DIP : Real;
      CTL_HTR_2_TMP_T1_DIP : Real;
      CTL_HTR_2_TMP_GN : Real;   // dword 480
      CTL_HTR_2_TMP_TI : Real;
      CTL_HTR_2_TMP_TD : Real;
      CTL_HTR_2_TMP_T1 : Real;
      CTL_HTR_1_MAX_PWR : Real;
      CTL_HTR_2_MAX_PWR : Real;
      CTL_MOB_FDR_VIB_GN : Real;
      CTL_MOB_FDR_VIB_TI : Real;
      CTL_MOB_FDR_VIB_TD : Real;   // dword 512
      CTL_MOB_FDR_VIB_T1 : Real;
      MCONST_LD_CL_1_MEAS_RNG : Real;
      CTL_PRS_GN : Real;
      CTL_PRS_TI : Real;
      CTL_PRS_TD : Real;
      CTL_PRS_T1 : Real;
      CTL_PRS_GN_HI : Real;
      CTL_PRS_TI_HI : Real;   // dword 544
      CTL_PRS_TD_HI : Real;
      CTL_PRS_T1_HI : Real;
      CTL_MLT_DRIFT_GN : Real;
      CTL_MLT_DRIFT_TI : Real;
      CTL_MLT_DRIFT_TD : Real;
      CTL_MLT_DRIFT_T1 : Real;
      MCONST_LD_CL_1_SMP_RNG : Real;
      PRS_CTRL_STD_ALG : Real;   // dword 576
      DIA_CTRL_STD_ALG : Real;
      HTR_1_CTRL_STD_ALG : Real;
      SPD_CTRL_STD_ALG : Real;
      CRUC_ROT_CTRL_STD_ALG : Real;
      MLT_TMP_CTRL_STD_ALG : Real;
      GRW_RTE_CTRL_STD_ALG : Real;
      MCONST_LD_CL_1_AVG_FILT : Real;
      ME_MAX_MLT_TMP : Real;   // dword 608
      FDG_MAX_HTR_1_PWR : Real;
      PD_V1_POS : Real;
      LIM_MLT_DRIFT_OFFS : Real;
      LIM_MLT_LVL_DEV : Real;
      LIM_XT_SPD : Real;
      LIM_XT_ROT : Real;
      LIM_CR_SPD : Real;
      LIM_CR_ROT : Real;   // dword 640
      LIM_SPD_DLY : Real;
      LIM_GAS_1_FLW : Real;
      LIM_GAS_2_FLW : Real;
      LIM_PRS : Real;
      LIM_GAS_FLW_DLY : Real;
      LIM_HTR_1_PWR : Real;
      LIM_HTR_2_PWR : Real;
      LIM_HTR_PWR_DLY : Real;   // dword 672
      LIM_HTR_1_RES : Real;
      LIM_HTR_2_RES : Real;
      LIM_MAG_1_CUR : Real;
      LIM_MAG_2_CUR : Real;
      LIM_MAG_DLY : Real;
      LIM_GRO : Real;
      LIM_GRO_DLY : Real;
      LIM_DIA_NECK_MIN : Real;   // dword 704
      LIM_DIA_NECK_DLY : Real;
      LIM_DIA_BODY_1 : Real;
      LIM_DIA_BODY_2 : Real;
      LIM_DIA_DLY : Real;
      LIM_AV_SPD_NE : Real;
      LIM_AV_SPD_BY1 : Real;
      LIM_AV_SPD_BY2 : Real;
      LIM_AV_SPD_DLY : Real;   // dword 736
      LIM_MLT_LVL : Real;
      LIM_MLT_LVL_DLY : Real;
      LIM_LEN_BODY1 : Real;
      LIM_MAG_1_RES : Real;
      LIM_MAG_2_RES : Real;
      LIM_THR_DEV : Real;
      MCONST_MLT_TMP_OFFS : Real;
      MCONST_ROT_DIR : Real;   // dword 768
      MCONST_DIA_CAL_P1 : Real;
      MCONST_DIA_CAL_P2 : Real;
      MCONST_DIA_2_CAL_P1 : Real;
      MCONST_DIA_2_CAL_P2 : Real;
      VAC_SEL_V2_PD : Real;
      VAC_SEL_V2_ME : Real;
      VAC_SEL_V2_DI : Real;
      VAC_SEL_V2_NE : Real;   // dword 800
      VAC_SEL_V2_SH : Real;
      VAC_SEL_V2_BY : Real;
      VAC_SEL_V2_EC : Real;
      VAC_SEL_V2_SD : Real;
      VAC_SEL_V2_RE : Real;
      MCONST_LIM_XTAL_UP : Real;
      MCONST_LIM_XTAL_DN : Real;
      MCONST_LIM_CR_UP : Real;   // dword 832
      MCONST_LIM_CR_DN : Real;
      MCONST_XT_ORB_LIM_NE : Real;
      MCONST_XT_ORB_LIM_SH : Real;
      MCONST_XT_ORB_LIM_BY : Real;
      MCONST_MLT_LVL_CAL : Real;
      MCONST_EMG_WAIT_TME : Real;
      MCONST_EMG_XT_LFT_DIST : Real;
      MCONST_EMG_CR_POS : Real;   // dword 864
      MCONST_EMG_XT_SPD : Real;
      MCONST_EMG_CR_SPD : Real;
      MCONST_XT_LD_CELL_CAL : Real;
      MCONST_DIA_MSR_MTH : Real;
      MCONST_MIN_AMT_MSR_PTS : Real;
      MCONST_MIN_LAT_XT_GRW : Real;
      MCONST_IMG_TRG_DLY : Real;
      MOB_FDR_DCK_PRG_CYC : Real;   // dword 896
      MOB_FDR_DCK_PRG_PRS : Real;
      MOB_FDR_DCK_PRG_TME : Real;
      MOB_FDR_DCK_FIN_PRS : Real;
      MOB_FDR_DCK_WAIT_TME : Real;
      MOB_FDR_DCK_LKT_TME : Real;
      MOB_FDR_DCK_MAX_LKR : Real;
      MOB_FDR_COOL_V24_ON : Real;
      MOB_FDR_SPARE_928 : Real;   // dword 928
      MOB_FDR_SPARE_932 : Real;
      MOB_FDR_UDCK_LKT_TME : Real;
      MOB_FDR_UDCK_MAX_PRS_DRP : Real;
      MOB_FDR_TUBE_COOL_STP : Real;
      MOB_FDR_TUBE_TRV_INC : Real;
      MOB_FDR_TUBE_COOL_DN_TME : Real;
      MCONST_MOB_FDR_LDC_CAL : Real;
      NE_MIN_LEN : Real;   // dword 960
      NE_MAX_LEN : Real;
      NE_STB_LEN : Real;
      NE_MAX_DEV_DIA : Real;
      NE_MAX_DEV_LAT_GRW : Real;
      SH_COEFFICIENT_A : Real;
      SH_COEFFICIENT_B : Real;
      SH_BY_TRS_MAX_DIA : Real;
      MCONST_V1_MAX_V2_1_CL : Real;   // dword 992
      MCONST_V2_1_DLY_TME : Real;
      MCONST_HTR_1_MAX_HOT_RES : Real;
      MCONST_HTR_1_MIN_HOT_RES : Real;
      MCONST_HTR_1_TMP_RES_MON : Real;
      MCONST_DST_CR_BOT_FNL : Real;
      DI_NE_REMLT_SPD : Real;
      ME_GAP_MLT_FNL : Real;
      RC_XT_LFT_TME : Real;   // dword 1024
      RC_XT_LFT_SPD : Real;
      RC_XT_COOL_DN_TME : Real;
      RC_XT_COOL_DN_TME_AR : Real;
      RC_FIN_PRS_PMP_DN : Real;
      BY_MLT_LVL_SFT_STR_LEN : Real;
      BY_MLT_LVL_SFT_LEN : Real;
      BY_MLT_LVL_SFT_OFFS_SPD : Real;
      SD_WAIT_UNTIL_VENT : Real;   // dword 1056
      BY_LEN_DIA_TMP_CTL_ON : Real;
      SD_WAIT_AFT_VENT : Real;
      ME_V21_OPEN : Real;
      DI_V21_OPEN : Real;
      NE_V21_OPEN : Real;
      SH_V21_OPEN : Real;
      BY_V21_OPEN : Real;
      RC_V21_OPEN : Real;   // dword 1088
      SH_MLT_LVL_SFT_STR_LEN : Real;
      SH_MLT_LVL_SFT_LEN : Real;
      SH_MLT_LVL_SFT_OFFS_SPD : Real;
      NE_MIN_XT_SPD : Real;
      NE_LEN_FLX : Real;
      SH_TRS_FLX : Real;
      MCONST_CR_ROT_TORQ_LIM : Real;
      ME_STD_DEV_FILL_LVL_HOP : Real;   // dword 1120
      ME_CALC_TME_STD_DEV : Real;
      HOP_FILL_LVL_DLY : Real;
      FDG_RTE_DLY : Real;
      CTL_FDG_RTE_OFF_LVL : Real;
      CTL_FDG_RTE_GN : Real;
      CTL_FDG_RTE_TI : Real;
      CTL_FDG_RTE_TD : Real;
      CTL_FDG_RTE_T1 : Real;   // dword 1152
      CTL_FDG_RTE_ON_DLY : Real;
      CTL_FDG_RTE_START_VAL : Real;
      CTL_LIM_FRQ_LOW : Real;
      CTL_LIM_FRQ_HI : Real;
      CTL_VIB_SET_P_ALM_DLY : Real;
      FDR_CUTE_WGT_DLY : Real;
      FDR_CUTE_WGT_RA : Real;
      MOB_FDR_DCK_ALM_TME1 : Real;   // dword 1184
      MOB_FDR_DCK_ALM_TME2 : Real;
      MOB_FDR_DCK_PRS_TRG1 : Real;
      MOB_FDR_DCK_PRS_TRG2 : Real;
      RE_STD_DEV_FILL_LVL_HOP : Real;
      RE_CALC_TME_STD_DEV : Real;
      CTL_AVG_GAP_OFFS_TF : Real;
      SET_GAP_OFFS_HL : Real;
      DI_MIN_HTR_1_PWR_LIM : Real;   // dword 1216
      DI_MAX_HTR_1_PWR_LIM : Real;
      SET_GAP_OFFS_LL : Real;
      SET_OFFS_SPEED_HL : Real;
      SET_OFFS_SPEED_LL : Real;
      MCONST_DIA_COR_MLT_LVL : Real;
      CTL_DIA_COR_SEL : Real;
      MCONST_DIA_COR_GAP_DEV : Real;
      MCONST_ANG_OF_PLX_SCAM : Real;   // dword 1248
      MCONST_CF_TO_RAD_PT_SCAM : Real;
      MCONST_CAL_CF_SCAM : Real;
      MCONST_CAL_RAD_PT_SCAM : Real;
      MCONST_CAL_MLT_LVL_SCAM : Real;
      EC_V21_OPEN : Real;
      SD_V21_OPEN : Real;
      SH_PWR_GAP_HTR_1 : Real;
      DI_PWR_GAP_HTR_1 : Real;   // dword 1280
      DI_PWR_DEC_HTR_1 : Real;
      SD_P1_GAS_BAL_V_OP : Real;
      MCONST_DST_LSR_MLT_LVL : Real;
      MCONST_CAM_1_INIT_RAD_PT : Real;
      MCONST_CAM_2_INIT_RAD_PT : Real;
      MCONST_SCAM_INIT_DIA : Real;
      SPARE_1308 : Real;
      SPARE_1312 : Real;   // dword 1312
      SPARE_1316 : Real;
      SPARE_1320 : Real;
      SPARE_1324 : Real;
      SPARE_1328 : Real;
      SPARE_1332 : Real;
      SPARE_1336 : Real;
      SPARE_1340 : Real;
   END_VAR
BEGIN
END_DATA_BLOCK

DATA_BLOCK "PAR_XT_SPD"   // DB11
{ S7_Optimized_Access := 'FALSE' }
VERSION : 0.0
BEGIN
END_DATA_BLOCK

DATA_BLOCK "PAR_XT_ROT"   // DB12
{ S7_Optimized_Access := 'FALSE' }
VERSION : 0.0
BEGIN
END_DATA_BLOCK

DATA_BLOCK "PAR_XT_POS"   // DB13
{ S7_Optimized_Access := 'FALSE' }
VERSION : 0.0
BEGIN
END_DATA_BLOCK

DATA_BLOCK "PAR_CR_SPD"   // DB14
{ S7_Optimized_Access := 'FALSE' }
VERSION : 0.0
BEGIN
END_DATA_BLOCK

DATA_BLOCK "PAR_CR_ROT"   // DB15
{ S7_Optimized_Access := 'FALSE' }
VERSION : 0.0
BEGIN
END_DATA_BLOCK

DATA_BLOCK "PAR_CR_POS"   // DB16
{ S7_Optimized_Access := 'FALSE' }
VERSION : 0.0
BEGIN
END_DATA_BLOCK

DATA_BLOCK "PAR_CRSPD_COEFF"   // DB17
{ S7_Optimized_Access := 'FALSE' }
VERSION : 0.0
BEGIN
END_DATA_BLOCK

DATA_BLOCK "PAR_CR_ROT_ON_TME"   // DB18
{ S7_Optimized_Access := 'FALSE' }
VERSION : 0.0
BEGIN
END_DATA_BLOCK

DATA_BLOCK "PAR_CR_ROT_OFF_TME"   // DB19
{ S7_Optimized_Access := 'FALSE' }
VERSION : 0.0
BEGIN
END_DATA_BLOCK

DATA_BLOCK "PAR_CR_ROT_OFFSET"   // DB20
{ S7_Optimized_Access := 'FALSE' }
VERSION : 0.0
BEGIN
END_DATA_BLOCK

DATA_BLOCK "PAR_FDR_VIB_FRQ"   // DB21
{ S7_Optimized_Access := 'FALSE' }
VERSION : 0.0
BEGIN
END_DATA_BLOCK

DATA_BLOCK "PAR_HTR_1_PWR"   // DB22
{ S7_Optimized_Access := 'FALSE' }
VERSION : 0.0
BEGIN
END_DATA_BLOCK

DATA_BLOCK "PAR_HTR_2_PWR"   // DB23
{ S7_Optimized_Access := 'FALSE' }
VERSION : 0.0
BEGIN
END_DATA_BLOCK

DATA_BLOCK "PAR_HTR_1_TMP"   // DB24
{ S7_Optimized_Access := 'FALSE' }
VERSION : 0.0
BEGIN
END_DATA_BLOCK

DATA_BLOCK "PAR_HTR_2_TMP"   // DB25
{ S7_Optimized_Access := 'FALSE' }
VERSION : 0.0
BEGIN
END_DATA_BLOCK

DATA_BLOCK "PAR_MAG_AV_CUR"   // DB26
{ S7_Optimized_Access := 'FALSE' }
VERSION : 0.0
BEGIN
END_DATA_BLOCK

DATA_BLOCK "PAR_MAG_RATIO_CUR"   // DB28
{ S7_Optimized_Access := 'FALSE' }
VERSION : 0.0
BEGIN
END_DATA_BLOCK

DATA_BLOCK "PAR_PRS"   // DB29
{ S7_Optimized_Access := 'FALSE' }
VERSION : 0.0
BEGIN
END_DATA_BLOCK

DATA_BLOCK "PAR_GAS_1_FLW"   // DB30
{ S7_Optimized_Access := 'FALSE' }
VERSION : 0.0
BEGIN
END_DATA_BLOCK

DATA_BLOCK "PAR_GAS_2_FLW"   // DB31
{ S7_Optimized_Access := 'FALSE' }
VERSION : 0.0
BEGIN
END_DATA_BLOCK

DATA_BLOCK "PAR_GAS_SUM_FLW"   // DB32
{ S7_Optimized_Access := 'FALSE' }
VERSION : 0.0
BEGIN
END_DATA_BLOCK

DATA_BLOCK "PAR_XT_DIA"   // DB33
{ S7_Optimized_Access := 'FALSE' }
VERSION : 0.0
BEGIN
END_DATA_BLOCK

DATA_BLOCK "PAR_AV_SPD"   // DB34
{ S7_Optimized_Access := 'FALSE' }
VERSION : 0.0
BEGIN
END_DATA_BLOCK

DATA_BLOCK "PAR_AV_SPD_DEV_1"   // DB35
{ S7_Optimized_Access := 'FALSE' }
VERSION : 0.0
BEGIN
END_DATA_BLOCK

DATA_BLOCK "PAR_AV_SPD_DEV_2"   // DB36
{ S7_Optimized_Access := 'FALSE' }
VERSION : 0.0
BEGIN
END_DATA_BLOCK

DATA_BLOCK "PAR_XT_GRO"   // DB37
{ S7_Optimized_Access := 'FALSE' }
VERSION : 0.0
BEGIN
END_DATA_BLOCK

DATA_BLOCK "PAR_MLT_TMP_1"   // DB38
{ S7_Optimized_Access := 'FALSE' }
VERSION : 0.0
BEGIN
END_DATA_BLOCK

DATA_BLOCK "PAR_MLT_LVL_INC"   // DB39
{ S7_Optimized_Access := 'FALSE' }
VERSION : 0.0
BEGIN
END_DATA_BLOCK

DATA_BLOCK "PAR_CTRL_DIA_GN"   // DB41
{ S7_Optimized_Access := 'FALSE' }
VERSION : 0.0
BEGIN
END_DATA_BLOCK

DATA_BLOCK "PAR_CTRL_DIA_TI"   // DB42
{ S7_Optimized_Access := 'FALSE' }
VERSION : 0.0
BEGIN
END_DATA_BLOCK

DATA_BLOCK "PAR_CTRL_DIA_TD"   // DB43
{ S7_Optimized_Access := 'FALSE' }
VERSION : 0.0
BEGIN
END_DATA_BLOCK

DATA_BLOCK "PAR_CTRL_DIA_T1"   // DB44
{ S7_Optimized_Access := 'FALSE' }
VERSION : 0.0
BEGIN
END_DATA_BLOCK

DATA_BLOCK "PAR_CTRL_DIA_TF"   // DB45
{ S7_Optimized_Access := 'FALSE' }
VERSION : 0.0
BEGIN
END_DATA_BLOCK

DATA_BLOCK "PAR_CTRL_GRO_GN"   // DB46
{ S7_Optimized_Access := 'FALSE' }
VERSION : 0.0
BEGIN
END_DATA_BLOCK

DATA_BLOCK "PAR_CTRL_GRO_TI"   // DB47
{ S7_Optimized_Access := 'FALSE' }
VERSION : 0.0
BEGIN
END_DATA_BLOCK

DATA_BLOCK "PAR_CTRL_GRO_TD"   // DB48
{ S7_Optimized_Access := 'FALSE' }
VERSION : 0.0
BEGIN
END_DATA_BLOCK

DATA_BLOCK "PAR_CTRL_GRO_T1"   // DB49
{ S7_Optimized_Access := 'FALSE' }
VERSION : 0.0
BEGIN
END_DATA_BLOCK

DATA_BLOCK "PAR_CTRL_GRO_TF"   // DB50
{ S7_Optimized_Access := 'FALSE' }
VERSION : 0.0
BEGIN
END_DATA_BLOCK

DATA_BLOCK "PAR_CTRL_AV_SPD_GN"   // DB51
{ S7_Optimized_Access := 'FALSE' }
VERSION : 0.0
BEGIN
END_DATA_BLOCK

DATA_BLOCK "PAR_CTRL_AV_SPD_TI"   // DB52
{ S7_Optimized_Access := 'FALSE' }
VERSION : 0.0
BEGIN
END_DATA_BLOCK

DATA_BLOCK "PAR_CTRL_AV_SPD_TD"   // DB53
{ S7_Optimized_Access := 'FALSE' }
VERSION : 0.0
BEGIN
END_DATA_BLOCK

DATA_BLOCK "PAR_CTRL_AV_SPD_T1"   // DB54
{ S7_Optimized_Access := 'FALSE' }
VERSION : 0.0
BEGIN
END_DATA_BLOCK

DATA_BLOCK "PAR_CTRL_AV_SPD_TF"   // DB55
{ S7_Optimized_Access := 'FALSE' }
VERSION : 0.0
BEGIN
END_DATA_BLOCK

DATA_BLOCK "PAR_CTRL_MLT_LVL_GN"   // DB56
{ S7_Optimized_Access := 'FALSE' }
VERSION : 0.0
BEGIN
END_DATA_BLOCK

DATA_BLOCK "PAR_CTRL_MLT_LVL_TI"   // DB57
{ S7_Optimized_Access := 'FALSE' }
VERSION : 0.0
BEGIN
END_DATA_BLOCK

DATA_BLOCK "PAR_CTRL_MLT_LVL_TD"   // DB58
{ S7_Optimized_Access := 'FALSE' }
VERSION : 0.0
BEGIN
END_DATA_BLOCK

DATA_BLOCK "PAR_CTRL_MLT_LVL_T1"   // DB59
{ S7_Optimized_Access := 'FALSE' }
VERSION : 0.0
BEGIN
END_DATA_BLOCK

DATA_BLOCK "PAR_CTRL_MLT_LVL_TF"   // DB60
{ S7_Optimized_Access := 'FALSE' }
VERSION : 0.0
BEGIN
END_DATA_BLOCK

DATA_BLOCK "PAR_CTRL_MLT_TMP_1_GN"   // DB61
{ S7_Optimized_Access := 'FALSE' }
VERSION : 0.0
BEGIN
END_DATA_BLOCK

DATA_BLOCK "PAR_CTRL_MLT_TMP_1_TI"   // DB62
{ S7_Optimized_Access := 'FALSE' }
VERSION : 0.0
BEGIN
END_DATA_BLOCK

DATA_BLOCK "PAR_CTRL_MLT_TMP_1_TD"   // DB63
{ S7_Optimized_Access := 'FALSE' }
VERSION : 0.0
BEGIN
END_DATA_BLOCK

DATA_BLOCK "PAR_CTRL_MLT_TMP_1_T1"   // DB64
{ S7_Optimized_Access := 'FALSE' }
VERSION : 0.0
BEGIN
END_DATA_BLOCK

DATA_BLOCK "PAR_CTRL_MLT_TMP_1_TF"   // DB65
{ S7_Optimized_Access := 'FALSE' }
VERSION : 0.0
BEGIN
END_DATA_BLOCK

DATA_BLOCK "PAR_CTRL_PRS_GN"   // DB66
{ S7_Optimized_Access := 'FALSE' }
VERSION : 0.0
BEGIN
END_DATA_BLOCK

DATA_BLOCK "PAR_CTRL_PRS_TI"   // DB67
{ S7_Optimized_Access := 'FALSE' }
VERSION : 0.0
BEGIN
END_DATA_BLOCK

DATA_BLOCK "PAR_CTRL_PRS_TD"   // DB68
{ S7_Optimized_Access := 'FALSE' }
VERSION : 0.0
BEGIN
END_DATA_BLOCK

DATA_BLOCK "PAR_CTRL_PRS_T1"   // DB69
{ S7_Optimized_Access := 'FALSE' }
VERSION : 0.0
BEGIN
END_DATA_BLOCK

DATA_BLOCK "PAR_CTRL_PRS_TF"   // DB70
{ S7_Optimized_Access := 'FALSE' }
VERSION : 0.0
BEGIN
END_DATA_BLOCK

DATA_BLOCK "PAR_CTRL_DIA_TMP_GN"   // DB71
{ S7_Optimized_Access := 'FALSE' }
VERSION : 0.0
BEGIN
END_DATA_BLOCK

DATA_BLOCK "PAR_CTRL_DIA_TMP_TI"   // DB72
{ S7_Optimized_Access := 'FALSE' }
VERSION : 0.0
BEGIN
END_DATA_BLOCK

DATA_BLOCK "PAR_XT_MEN"   // DB73
{ S7_Optimized_Access := 'FALSE' }
VERSION : 0.0
BEGIN
END_DATA_BLOCK

DATA_BLOCK "PAR_CTRL_DIA_TMP_TD"   // DB74
{ S7_Optimized_Access := 'FALSE' }
VERSION : 0.0
BEGIN
END_DATA_BLOCK

DATA_BLOCK "PAR_CR_CHARGE_WGT"   // DB75
{ S7_Optimized_Access := 'FALSE' }
VERSION : 0.0
BEGIN
END_DATA_BLOCK

DATA_BLOCK "PAR_CR_DIA"   // DB76
{ S7_Optimized_Access := 'FALSE' }
VERSION : 0.0
BEGIN
END_DATA_BLOCK

DATA_BLOCK "PAR_CR_FILL_LEVEL"   // DB77
{ S7_Optimized_Access := 'FALSE' }
VERSION : 0.0
BEGIN
END_DATA_BLOCK

DATA_BLOCK "PAR_CTRL_DIA_TMP_T1"   // DB78
{ S7_Optimized_Access := 'FALSE' }
VERSION : 0.0
BEGIN
END_DATA_BLOCK

DATA_BLOCK "PAR_TMP_COEFF_1"   // DB80
{ S7_Optimized_Access := 'FALSE' }
VERSION : 0.0
BEGIN
END_DATA_BLOCK

DATA_BLOCK "PAR_TMP_COEFF_2"   // DB81
{ S7_Optimized_Access := 'FALSE' }
VERSION : 0.0
BEGIN
END_DATA_BLOCK

DATA_BLOCK "PAR_PWR_COEFF_1"   // DB82
{ S7_Optimized_Access := 'FALSE' }
VERSION : 0.0
BEGIN
END_DATA_BLOCK

DATA_BLOCK "PAR_PWR_COEFF_2"   // DB83
{ S7_Optimized_Access := 'FALSE' }
VERSION : 0.0
BEGIN
END_DATA_BLOCK

DATA_BLOCK "PAR_CAM_THR"   // DB86
{ S7_Optimized_Access := 'FALSE' }
VERSION : 0.0
BEGIN
END_DATA_BLOCK

DATA_BLOCK "PAR_CAM_WIN_SIZE_H"   // DB87
{ S7_Optimized_Access := 'FALSE' }
VERSION : 0.0
BEGIN
END_DATA_BLOCK

DATA_BLOCK "PAR_CAM_WIN_SIZE_V"   // DB88
{ S7_Optimized_Access := 'FALSE' }
VERSION : 0.0
BEGIN
END_DATA_BLOCK

DATA_BLOCK "PAR_CAM_WIN_POS_H"   // DB89
{ S7_Optimized_Access := 'FALSE' }
VERSION : 0.0
BEGIN
END_DATA_BLOCK

DATA_BLOCK "PAR_CAM_WIN_POS_V"   // DB90
{ S7_Optimized_Access := 'FALSE' }
VERSION : 0.0
BEGIN
END_DATA_BLOCK

DATA_BLOCK "PAR_TME"   // DB91
{ S7_Optimized_Access := 'FALSE' }
VERSION : 0.0
BEGIN
END_DATA_BLOCK

DATA_BLOCK "PAR_X_VALUES_1"   // DB92
{ S7_Optimized_Access := 'FALSE' }
VERSION : 0.0
BEGIN
END_DATA_BLOCK

DATA_BLOCK "PAR_X_VALUES_2"   // DB93
{ S7_Optimized_Access := 'FALSE' }
VERSION : 0.0
BEGIN
END_DATA_BLOCK

DATA_BLOCK "PAR_X_VALUES_3"   // DB94
{ S7_Optimized_Access := 'FALSE' }
VERSION : 0.0
BEGIN
END_DATA_BLOCK

DATA_BLOCK "PAR_X_VALUES_4"   // DB95
{ S7_Optimized_Access := 'FALSE' }
VERSION : 0.0
BEGIN
END_DATA_BLOCK

DATA_BLOCK "PAR_X_VALUES_5"   // DB96
{ S7_Optimized_Access := 'FALSE' }
VERSION : 0.0
BEGIN
END_DATA_BLOCK

DATA_BLOCK "PAR_X_VALUES_6"   // DB97
{ S7_Optimized_Access := 'FALSE' }
VERSION : 0.0
BEGIN
END_DATA_BLOCK

DATA_BLOCK "PAR_X_VALUES_7"   // DB98
{ S7_Optimized_Access := 'FALSE' }
VERSION : 0.0
BEGIN
END_DATA_BLOCK

DATA_BLOCK "PAR_X_VALUES_8"   // DB99
{ S7_Optimized_Access := 'FALSE' }
VERSION : 0.0
BEGIN
END_DATA_BLOCK

DATA_BLOCK "PAR_X_VALUES_9"   // DB100
{ S7_Optimized_Access := 'FALSE' }
VERSION : 0.0
BEGIN
END_DATA_BLOCK

DATA_BLOCK "PAR_X_VALUES_10"   // DB101
{ S7_Optimized_Access := 'FALSE' }
VERSION : 0.0
BEGIN
END_DATA_BLOCK

DATA_BLOCK "PAR_AV_CRUC_ROT"   // DB102
{ S7_Optimized_Access := 'FALSE' }
VERSION : 0.0
BEGIN
END_DATA_BLOCK

DATA_BLOCK "PAR_AV_CRUC_ROT_DEV_1"   // DB103
{ S7_Optimized_Access := 'FALSE' }
VERSION : 0.0
BEGIN
END_DATA_BLOCK

DATA_BLOCK "PAR_AV_CRUC_ROT_DEV_2"   // DB104
{ S7_Optimized_Access := 'FALSE' }
VERSION : 0.0
BEGIN
END_DATA_BLOCK

DATA_BLOCK "PAR_CTRL_AV_CRUC_ROT_GN"   // DB105
{ S7_Optimized_Access := 'FALSE' }
VERSION : 0.0
BEGIN
END_DATA_BLOCK

DATA_BLOCK "PAR_CTRL_AV_CRUC_ROT_TI"   // DB106
{ S7_Optimized_Access := 'FALSE' }
VERSION : 0.0
BEGIN
END_DATA_BLOCK

DATA_BLOCK "PAR_CTRL_AV_CRUC_ROT_TD"   // DB107
{ S7_Optimized_Access := 'FALSE' }
VERSION : 0.0
BEGIN
END_DATA_BLOCK

DATA_BLOCK "PAR_CTRL_AV_CRUC_ROT_T1"   // DB108
{ S7_Optimized_Access := 'FALSE' }
VERSION : 0.0
BEGIN
END_DATA_BLOCK

DATA_BLOCK "PAR_CR_ROT_RP_TME_UP"   // DB109
{ S7_Optimized_Access := 'FALSE' }
VERSION : 0.0
BEGIN
END_DATA_BLOCK

DATA_BLOCK "PAR_CR_ROT_RP_TME_DN"   // DB110
{ S7_Optimized_Access := 'FALSE' }
VERSION : 0.0
BEGIN
END_DATA_BLOCK

DATA_BLOCK "PAR_CAM_SET_OUT_RAD"   // DB111
{ S7_Optimized_Access := 'FALSE' }
VERSION : 0.0
BEGIN
END_DATA_BLOCK

DATA_BLOCK "PAR_CAM_SET_IN_RAD"   // DB112
{ S7_Optimized_Access := 'FALSE' }
VERSION : 0.0
BEGIN
END_DATA_BLOCK

DATA_BLOCK "PAR_CAM_SET_SEQ_STR_AGL"   // DB113
{ S7_Optimized_Access := 'FALSE' }
VERSION : 0.0
BEGIN
END_DATA_BLOCK

DATA_BLOCK "PAR_CAM_SET_SEQ_STP_AGL"   // DB114
{ S7_Optimized_Access := 'FALSE' }
VERSION : 0.0
BEGIN
END_DATA_BLOCK

DATA_BLOCK "PAR_X_VALUES_11"   // DB115
{ S7_Optimized_Access := 'FALSE' }
VERSION : 0.0
BEGIN
END_DATA_BLOCK

DATA_BLOCK "PM_TLU_PWR_SPL_DATA_BUF"   // DB127
{ S7_Optimized_Access := 'FALSE' }
VERSION : 0.0
// --------------------------------------------------------------------------------
//     program     :    PM_TLU_PWR_SPL_DATA_BUF
//     description :    data block buffer in-out-data of TLU power supply
//                            
//     name        :    G. Eibelsh鋟ser
//     date        :    16.04.2012
// 
//     revision    :   
//     name        :    
//     date        :   
//  
//                     (c)PVA TePla AG
//     --------------------------------------------------------------------------------
   VAR
      TLU_CTRL_IN : Struct   // TLU_CTRL Input data
         CUR_ACT_L : Byte;   // Data byte 0 Strom Istwert (first byte offset = 0)
         CUR_ACT_H : Byte;   // Data byte 1
         VLT_ACT_L : Byte;   // Data byte 2 Spannung Istwert
         VLT_ACT_H : Byte;   // Data byte 3
         STA_1_L : Byte;   // Data byte 4 Status 1
         STA_1_H : Byte;   // Data byte 5
         PWR_ACT_L : Byte;   // Data byte 6 Leistung Istwert
         PWR_ACT_H : Byte;   // Data byte 7
         FLT_MEM1_L : Byte;   // Data byte 8 Fehlerspeicher 1
         FLT_MEM1_H : Byte;   // Data byte 9
         FLT_MEM2_L : Byte;   // Data byte 10 Fehlerspeicher 2
         FLT_MEM2_H : Byte;   // Data byte 11
         FLT_1_L : Byte;   // Data byte 12 Fehler aktuell 1
         FLT_1_H : Byte;   // Data byte 13
         FLT_2_L : Byte;   // Data byte 14 Fehler aktuell 2
         FLT_2_H : Byte;   // Data byte 15
         CUR_NEN_L : Byte;   // Data byte 16 Strom Nennwert
         CUR_NEN_H : Byte;   // Data byte 17
         VLT_NEN_L : Byte;   // Data byte 18 Spannung Nennwert
         VLT_NEN_H : Byte;   // Data byte 19
         PWR_NEN_L : Byte;   // Data byte 20 Leistung Nennwert
         PWR_NEN_H : Byte;   // Data byte 21
         STA_2_L : Byte;   // Data byte 22 Status 2
         STA_2_H : Byte;   // Data byte 23
         ENRJ_1_L : Byte;   // Data byte 24 Energiez鋒ler 1
         ENRJ_1_H : Byte;   // Data byte 25
         ENRJ_2_L : Byte;   // Data byte 26 Energiez鋒ler 2
         ENRJ_2_H : Byte;   // Data byte 27
         ENRJ_3_L : Byte;   // Data byte 28 Energiez鋒ler 3
         ENRJ_3_H : Byte;   // Data byte 29
         PLS_L : Byte;   // Data byte 30 Pulsperiode
         PLS_H : Byte;   // Data byte 31
         PRESC_L : Byte;   // Data byte 32 Prescaler
         PRESC_H : Byte;   // Data byte 33
         FIRM_L : Byte;   // Data byte 34 Firmware
         FIRM_H : Byte;   // Data byte 35
      END_STRUCT;
      TLU_CTRL_OUT : Struct   // TLU_CTRL Output data
         CUR_SET_L : Byte;   // Data byte 0 Strom Sollwert (first byte offset = 36)
         CUR_SET_H : Byte;   // Data byte 1
         VLT_SET_L : Byte;   // Data byte 2 Spannung Sollwert
         VLT_SET_H : Byte;   // Data byte 3
         CTRL_1_L : Byte;   // Data byte 4 Steuerwort
         CTRL_1_H : Byte;   // Data byte 5
         PWR_SET_L : Byte;   // Data byte 6 Leistung Sollwert
         PWR_SET_H : Byte;   // Data byte 7
         PLS_PER_L : Byte;   // Data byte 8 Pulsperiode
         PLS_PER_H : Byte;   // Data byte 9
         PLS_WDT_L : Byte;   // Data byte 10 Pulsweite ein
         PLS_WDT_H : Byte;   // Data byte 11
         R_MIN_L : Byte;   // Data byte 12 R min???
         R_MIN_H : Byte;   // Data byte 13
         DELTA_U_L : Byte;   // Data byte 14 delta U???
         DELTA_U_H : Byte;   // Data byte 15
         PLS_PAK_L : Byte;   // Data byte 16 Puls je Packet
         PLS_PAK_H : Byte;   // Data byte 17
         PLS_PP_L : Byte;   // Data byte 18 PulsPacketPause
         PLS_PP_H : Byte;   // Data byte 19
         RI_SET_L : Byte;   // Data byte 20 Ri Sollwert???
         RI_SET_H : Byte;   // Data byte 21
         IWI_SET_L : Byte;   // Data byte 22 Iwi Sollwert???
         IWI_SET_H : Byte;   // Data byte 23
      END_STRUCT;
   END_VAR
BEGIN
END_DATA_BLOCK

DATA_BLOCK "APC"   // DB128
{ S7_Optimized_Access := 'FALSE' }
VERSION : 0.0
// --------------------------------------------------------------------------------
//     program     :   APC
//     description :   global APC variables       
//     name        :   G. Eibelsh鋟ser
//     date        :   27.10.2007
//     
//     revision    :   
//     name        :   
//     date        :    
//  
//                     (c)PVA TePla AG       
//     --------------------------------------------------------------------------------
   VAR
      AUTOMATIC : Bool;   // FALSE = MANUAL, TRUE = AUTOMATIC
      CONT : Bool;   // APC continue flag, switch to next step if continue enabled
      HOLD : Bool;   // APC hold flag, set sequence to hold mode for test
      SINGLE : Bool;   // APC sigle flag, sigle step in hold mode
      RESUME : Bool;   // APC resume flag, resume sequence in hold mode
      JUMP : Bool;   // APC jump flag, force sequence to next step in hold mode
      BLK : Bool;   // APC blink signal 1sec on 1sec off
      PD_WITH_ME : Bool;   // APC melting is started after pump down
      PNBDY : Bool;   // new body, values for 2nd body saved
      BYRST : Bool;   // body restart, seq. for 2nd body active
      SUTDN : Bool;   // endcone with shut down
      CALC_LEN2 : Bool;   // new length for 2nd body has to be calc.
      LEN2_CALC : Bool;   // new lenght for 2nd body was calc.
      RE_WHILE_BY : Bool;   // removal was started while body was active
      MOVE_CRUC_INTO_DIP_POS : Bool;   // request flag to move body into dip position
      STATUS : Int;   // activ APC status
      REQUEST : Int;   // requested APC status
      OP_MSG : Int;   // actual operator message process phases --------------
      IDLE : Int;   // APC #0 of idle mode
      CHARGING : Int;   // APC #1 of charging mode
      PUMP_DOWN : Int;   // APC #2 of pump down mode
      MELTING : Int;   // APC #3 of melting mode
      DIPPING : Int;   // APC #4 of dipping mode
      NECK : Int;   // APC #5 of neck mode
      SHOULDER : Int;   // APC #6 of shoulder mode
      BODY : Int;   // APC #7 of body mode
      ENDCONE : Int;   // APC #8 of endcone mode
      SHUT_DOWN : Int;   // APC #9 of shut down mode
      REMOVAL : Int;   // APC #10 of removal mode
      EMG : Int;   // APC #11 of emergency separation mode machine state -------------
      STATE_STD_BY : Int;   // APC #1 of state standby
      STATE_SERV : Int;   // APC #2 of state service
      STATE_RUN : Int;   // APC #3 of state process run
      STATE_VAC_TEST : Int;   // APC #4 of state vacuum test without melting
      STATE_LOADING : Int;   // APC #5 of state loading
      STATE_MAINTENANCE : Int;   // APC #6 of state maintenance
      STATE_ENGINEERING : Int;   // APC #7 of state engineering
      STATE_BAKE_OUT : Int;   // APC #8 of state bake out
      TI : Array[0..7] of Int;
      LTI : Array[0..3] of DInt;
      ACT_TME_TOT : DInt;   // total time
      ACT_TME_PROC : DInt;   // process time (for each phase)
      ACT_TME_STE : DInt;   // step time (till end of step)
   END_VAR
BEGIN
END_DATA_BLOCK

